LIN {X 0,Y 129.318,Z 434.565,A -85,B 0,C 180,E1 -25427.406,E2 -25427.406} C_VEL
LIN {X 0,Y 134.78,Z 442.453,A -85,B 0,C 180,E1 -25430.686,E2 -25430.686} C_VEL
LIN {X 0,Y 140.996,Z 452.81,A -85,B 0,C 180,E1 -25434.022,E2 -25434.022} C_VEL
LIN {X 0,Y 146.703,Z 463.984,A -85,B 0,C 180,E1 -25436.807,E2 -25436.807} C_VEL
LIN {X 0,Y 149.634,Z 472.659,A -85,B 0,C 180,E1 -25438.294,E2 -25438.294} C_VEL
LIN {X 0,Y 146.442,Z 521.623,A -85,B 0,C 180,E1 -25440.39,E2 -25440.39} C_VEL
LIN {X 0,Y 144.723,Z 534.957,A -85,B 0,C 180,E1 -25441.401,E2 -25441.401} C_VEL
LIN {X 0,Y 142.363,Z 547.629,A -85,B 0,C 180,E1 -25442.871,E2 -25442.871} C_VEL
LIN {X 0,Y 139.472,Z 559.922,A -85,B 0,C 180,E1 -25444.918,E2 -25444.918} C_VEL
LIN {X 0,Y 136.356,Z 570.543,A -85,B 0,C 180,E1 -25447.259,E2 -25447.259} C_VEL
LIN {X 0,Y 133.114,Z 580.026,A -85,B 0,C 180,E1 -25449.929,E2 -25449.929} C_VEL
LIN {X 0,Y 129.657,Z 589.7,A -85,B 0,C 180,E1 -25453.466,E2 -25453.466} C_VEL
LIN {X 0,Y 126.749,Z 597.618,A -85,B 0,C 180,E1 -25457.185,E2 -25457.185} C_VEL
LIN {X 0,Y 123.714,Z 605.371,A -85,B 0,C 180,E1 -25461.835,E2 -25461.835} C_VEL
LIN {X 0,Y 121.559,Z 611.578,A -85,B 0,C 180,E1 -25466.685,E2 -25466.685} C_VEL
LIN {X 0,Y 120.174,Z 616.507,A -85,B 0,C 180,E1 -25471.675,E2 -25471.675} C_VEL
LIN {X 0,Y 119.203,Z 620.325,A -85,B 0,C 180,E1 -25476.771,E2 -25476.771} C_VEL
LIN {X 0,Y 118.82,Z 622.302,A -85,B 0,C 180,E1 -25480.22,E2 -25480.22} C_VEL
LIN {X 0,Y 118.766,Z 623.841,A -85,B 0,C 180,E1 -25483.691,E2 -25483.691} C_VEL
LIN {X 0,Y 119.319,Z 625.43,A -85,B 0,C 180,E1 -25489.54,E2 -25489.54} C_VEL
LIN {X 0,Y 120.253,Z 625.873,A -85,B 0,C 180,E1 -25494.147,E2 -25494.147} C_VEL
LIN {X 0,Y 121.437,Z 625.705,A -85,B 0,C 180,E1 -25497.579,E2 -25497.579} C_VEL
LIN {X 0,Y 123.02,Z 625.088,A -85,B 0,C 180,E1 -25501.026,E2 -25501.026} C_VEL
LIN {X 0,Y 124.883,Z 624.1,A -85,B 0,C 180,E1 -25504.246,E2 -25504.246} C_VEL
LIN {X 0,Y 127.173,Z 622.663,A -85,B 0,C 180,E1 -25507.435,E2 -25507.435} C_VEL
LIN {X 0,Y 131.368,Z 619.573,A -85,B 0,C 180,E1 -25512.044,E2 -25512.044} C_VEL
LIN {X 0,Y 136.162,Z 615.452,A -85,B 0,C 180,E1 -25516.268,E2 -25516.268} C_VEL
LIN {X 0,Y 141.896,Z 609.877,A -85,B 0,C 180,E1 -25520.311,E2 -25520.311} C_VEL
LIN {X 0,Y 147.954,Z 603.18,A -85,B 0,C 180,E1 -25523.852,E2 -25523.852} C_VEL
LIN {X 0,Y 153.971,Z 595.672,A -85,B 0,C 180,E1 -25526.788,E2 -25526.788} C_VEL
LIN {X 0,Y 159.544,Z 587.649,A -85,B 0,C 180,E1 -25529.199,E2 -25529.199} C_VEL
LIN {X 0,Y 165.169,Z 578.312,A -85,B 0,C 180,E1 -25531.351,E2 -25531.351} C_VEL
LIN {X 0,Y 170.467,Z 567.735,A -85,B 0,C 180,E1 -25533.211,E2 -25533.211} C_VEL
LIN {X 0,Y 174.935,Z 556.816,A -85,B 0,C 180,E1 -25534.676,E2 -25534.676} C_VEL
LIN {X 0,Y 179.164,Z 543.992,A -85,B 0,C 180,E1 -25535.89,E2 -25535.89} C_VEL
LIN {X 0,Y 182.11,Z 531.516,A -85,B 0,C 180,E1 -25536.711,E2 -25536.711} C_VEL
LIN {X 0,Y 184.136,Z 518.177,A -85,B 0,C 180,E1 -25537.258,E2 -25537.258} C_VEL
LIN {X 0,Y 185.4,Z 503.746,A -85,B 0,C 180,E1 -25537.724,E2 -25537.724} C_VEL
LIN {X 0,Y 181.912,Z 495.534,A -85,B 0,C 180,E1 -25540.462,E2 -25540.462} C_VEL
LIN {X 0,Y 178.893,Z 489.105,A -85,B 0,C 180,E1 -25543.103,E2 -25543.103} C_VEL
LIN {X 0,Y 175.604,Z 483.621,A -85,B 0,C 180,E1 -25546.287,E2 -25546.287} C_VEL
LIN {X 0,Y 173.351,Z 479.892,A -85,B 0,C 180,E1 -25548.853,E2 -25548.853} C_VEL
LIN {X 0,Y 171.062,Z 476.076,A -85,B 0,C 180,E1 -25552.03,E2 -25552.03} C_VEL
LIN {X 0,Y 168.902,Z 472.452,A -85,B 0,C 180,E1 -25555.974,E2 -25555.974} C_VEL
LIN {X 0,Y 168.299,Z 471.765,A -85,B 0,C 180,E1 -25557.306,E2 -25557.306} C_VEL
LIN {X 0,Y 166.803,Z 469.612,A -85,B 0,C 180,E1 -25562.415,E2 -25562.415} C_VEL
LIN {X 0,Y 166.469,Z 469.381,A -85,B 0,C 180,E1 -25568.011,E2 -25568.011} C_VEL
LIN {X 0,Y 168.639,Z 472.395,A -85,B 0,C 180,E1 -25576.378,E2 -25576.378} C_VEL
LIN {X 0,Y 170.598,Z 475.906,A -85,B 0,C 180,E1 -25580.183,E2 -25580.183} C_VEL
LIN {X 0,Y 171.488,Z 476.948,A -85,B 0,C 180,E1 -25581.499,E2 -25581.499} C_VEL
LIN {X 0,Y 174.003,Z 481.404,A -85,B 0,C 180,E1 -25584.839,E2 -25584.839} C_VEL
LIN {X 0,Y 176.64,Z 486.542,A -85,B 0,C 180,E1 -25587.76,E2 -25587.76} C_VEL
LIN {X 0,Y 179.778,Z 493.205,A -85,B 0,C 180,E1 -25590.771,E2 -25590.771} C_VEL
LIN {X 0,Y 183.644,Z 502.498,A -85,B 0,C 180,E1 -25594.035,E2 -25594.035} C_VEL
LIN {X 0,Y 185.144,Z 506.515,A -85,B 0,C 180,E1 -25595.205,E2 -25595.205} C_VEL
LIN {X 0,Y 183.231,Z 526.342,A -85,B 0,C 180,E1 -25595.88,E2 -25595.88} C_VEL
LIN {X 0,Y 180.741,Z 539.674,A -85,B 0,C 180,E1 -25596.566,E2 -25596.566} C_VEL
LIN {X 0,Y 177.685,Z 550.971,A -85,B 0,C 180,E1 -25597.424,E2 -25597.424} C_VEL
LIN {X 0,Y 173.234,Z 563.127,A -85,B 0,C 180,E1 -25598.654,E2 -25598.654} C_VEL
LIN {X 0,Y 168.106,Z 574.487,A -85,B 0,C 180,E1 -25600.275,E2 -25600.275} C_VEL
LIN {X 0,Y 162.509,Z 584.748,A -85,B 0,C 180,E1 -25602.219,E2 -25602.219} C_VEL
LIN {X 0,Y 157.267,Z 593.136,A -85,B 0,C 180,E1 -25604.358,E2 -25604.358} C_VEL
LIN {X 0,Y 150.468,Z 602.273,A -85,B 0,C 180,E1 -25607.372,E2 -25607.372} C_VEL
LIN {X 0,Y 144.164,Z 609.633,A -85,B 0,C 180,E1 -25610.675,E2 -25610.675} C_VEL
LIN {X 0,Y 138.227,Z 615.973,A -85,B 0,C 180,E1 -25614.644,E2 -25614.644} C_VEL
LIN {X 0,Y 133.531,Z 620.248,A -85,B 0,C 180,E1 -25618.245,E2 -25618.245} C_VEL
LIN {X 0,Y 129.165,Z 623.859,A -85,B 0,C 180,E1 -25622.453,E2 -25622.453} C_VEL
LIN {X 0,Y 125.462,Z 626.488,A -85,B 0,C 180,E1 -25626.915,E2 -25626.915} C_VEL
LIN {X 0,Y 121.969,Z 628.597,A -85,B 0,C 180,E1 -25633.257,E2 -25633.257} C_VEL
LIN {X 0,Y 119.96,Z 629.091,A -85,B 0,C 180,E1 -25639.878,E2 -25639.878} C_VEL
LIN {X 0,Y 119.462,Z 628.772,A -85,B 0,C 180,E1 -25643.244,E2 -25643.244} C_VEL
LIN {X 0,Y 119.228,Z 628.073,A -85,B 0,C 180,E1 -25646.622,E2 -25646.622} C_VEL
LIN {X 0,Y 119.292,Z 626.945,A -85,B 0,C 180,E1 -25650.001,E2 -25650.001} C_VEL
LIN {X 0,Y 119.221,Z 625.38,A -85,B 0,C 180,E1 -25653.38,E2 -25653.38} C_VEL
LIN {X 0,Y 119.525,Z 622.215,A -85,B 0,C 180,E1 -25658.454,E2 -25658.454} C_VEL
LIN {X 0,Y 120.525,Z 617.966,A -85,B 0,C 180,E1 -25663.489,E2 -25663.489} C_VEL
LIN {X 0,Y 122.565,Z 611.486,A -85,B 0,C 180,E1 -25669.252,E2 -25669.252} C_VEL
LIN {X 0,Y 125.294,Z 604.381,A -85,B 0,C 180,E1 -25673.996,E2 -25673.996} C_VEL
LIN {X 0,Y 128.645,Z 595.462,A -85,B 0,C 180,E1 -25678.556,E2 -25678.556} C_VEL
LIN {X 0,Y 129.744,Z 592.221,A -85,B 0,C 180,E1 -25679.96,E2 -25679.96} C_VEL
LIN {X 0,Y 130.741,Z 588.009,A -85,B 0,C 180,E1 -25681.699,E2 -25681.699} C_VEL
LIN {X 0,Y 130.735,Z 580.813,A -85,B 0,C 180,E1 -25684.674,E2 -25684.674} C_VEL
LIN {X 0,Y 130.793,Z 573.141,A -85,B 0,C 180,E1 -25687.438,E2 -25687.438} C_VEL
LIN {X 0,Y 131.839,Z 568.125,A -85,B 0,C 180,E1 -25688.78,E2 -25688.78} C_VEL
LIN {X 0,Y 134.682,Z 558.276,A -85,B 0,C 180,E1 -25690.713,E2 -25690.713} C_VEL
LIN {X 0,Y 137.347,Z 546.808,A -85,B 0,C 180,E1 -25692.439,E2 -25692.439} C_VEL
LIN {X 0,Y 139.629,Z 533.737,A -85,B 0,C 180,E1 -25693.795,E2 -25693.795} C_VEL
LIN {X 0,Y 141.126,Z 520.65,A -85,B 0,C 180,E1 -25694.629,E2 -25694.629} C_VEL
LIN {X 0,Y 143.948,Z 477.532,A -85,B 0,C 180,E1 -25696.505,E2 -25696.505} C_VEL
LIN {X 0,Y 139.603,Z 464.581,A -85,B 0,C 180,E1 -25698.949,E2 -25698.949} C_VEL
LIN {X 0,Y 136.315,Z 456.813,A -85,B 0,C 180,E1 -25700.824,E2 -25700.824} C_VEL
LIN {X 0,Y 131.62,Z 448.624,A -85,B 0,C 180,E1 -25703.541,E2 -25703.541} C_VEL
LIN {X 0,Y 127.404,Z 442.333,A -85,B 0,C 180,E1 -25706.19,E2 -25706.19} C_VEL
LIN {X 0,Y 124.865,Z 438.651,A -85,B 0,C 180,E1 -25707.944,E2 -25707.944} C_VEL
LIN {X 0,Y 121.967,Z 434.646,A -85,B 0,C 180,E1 -25710.108,E2 -25710.108} C_VEL
LIN {X 0,Y 119.651,Z 431.734,A -85,B 0,C 180,E1 -25711.972,E2 -25711.972} C_VEL
LIN {X 0,Y 118.813,Z 430.199,A -85,B 0,C 180,E1 -25712.74,E2 -25712.74} C_VEL
LIN {X 0,Y 116.336,Z 428.193,A -85,B 0,C 180,E1 -25714.876,E2 -25714.876} C_VEL
LIN {X 0,Y 115.061,Z 425.271,A -85,B 0,C 180,E1 -25716.596,E2 -25716.596} C_VEL
LIN {X 0,Y 114.987,Z 424.725,A -85,B 0,C 180,E1 -25717.686,E2 -25717.686} C_VEL
LIN {X 0,Y 114.999,Z 424.63,A -85,B 0,C 180,E1 -25722.207,E2 -25722.207} C_VEL
LIN {X 0,Y 115.248,Z 424.589,A -85,B 0,C 180,E1 -25727.343,E2 -25727.343} C_VEL
LIN {X 0,Y 115.361,Z 424.586,A -85,B 0,C 180,E1 -25733.001,E2 -25733.001} C_VEL
LIN {X 0,Y 115.992,Z 424.48,A -85,B 0,C 180,E1 -25740,E2 -25740} C_VEL
LIN {X 0,Y 115.365,Z 424.614,A -85,B 0,C 180,E1 -25746.998,E2 -25746.998} C_VEL
LIN {X 0,Y 115.208,Z 424.575,A -85,B 0,C 180,E1 -25752.567,E2 -25752.567} C_VEL
LIN {X 0,Y 115.005,Z 424.657,A -85,B 0,C 180,E1 -25757.791,E2 -25757.791} C_VEL
LIN {X 0,Y 114.946,Z 424.613,A -85,B 0,C 180,E1 -25763.491,E2 -25763.491} C_VEL
LIN {X 0,Y 114.862,Z 424.646,A -85,B 0,C 180,E1 -25771.062,E2 -25771.062} C_VEL
LIN {X 0,Y 114.893,Z 424.978,A -85,B 0,C 180,E1 -25776.14,E2 -25776.14} C_VEL
LIN {X 0,Y 115.165,Z 426.179,A -85,B 0,C 180,E1 -25777.121,E2 -25777.121} C_VEL
LIN {X 0,Y 116.635,Z 428.622,A -85,B 0,C 180,E1 -25778.672,E2 -25778.672} C_VEL
LIN {X 0,Y 118.86,Z 430.392,A -85,B 0,C 180,E1 -25780.572,E2 -25780.572} C_VEL
LIN {X 0,Y 120.727,Z 433.562,A -85,B 0,C 180,E1 -25782.221,E2 -25782.221} C_VEL
LIN {X 0,Y 122.798,Z 435.75,A -85,B 0,C 180,E1 -25783.788,E2 -25783.788} C_VEL
LIN {X 0,Y 125.433,Z 439.341,A -85,B 0,C 180,E1 -25785.707,E2 -25785.707} C_VEL
LIN {X 0,Y 131.141,Z 447.832,A -85,B 0,C 180,E1 -25789.424,E2 -25789.424} C_VEL
LIN {X 0,Y 136.678,Z 457.327,A -85,B 0,C 180,E1 -25792.621,E2 -25792.621} C_VEL
LIN {X 0,Y 141.992,Z 468.051,A -85,B 0,C 180,E1 -25795.435,E2 -25795.435} C_VEL
LIN {X 0,Y 144.087,Z 474.399,A -85,B 0,C 180,E1 -25796.594,E2 -25796.594} C_VEL
LIN {X 0,Y 140.883,Z 521.133,A -85,B 0,C 180,E1 -25798.623,E2 -25798.623} C_VEL
LIN {X 0,Y 139.202,Z 534.074,A -85,B 0,C 180,E1 -25799.594,E2 -25799.594} C_VEL
LIN {X 0,Y 136.886,Z 546.091,A -85,B 0,C 180,E1 -25800.956,E2 -25800.956} C_VEL
LIN {X 0,Y 134.056,Z 558.251,A -85,B 0,C 180,E1 -25802.952,E2 -25802.952} C_VEL
LIN {X 0,Y 130.727,Z 569.365,A -85,B 0,C 180,E1 -25805.377,E2 -25805.377} C_VEL
LIN {X 0,Y 127.21,Z 579.081,A -85,B 0,C 180,E1 -25808.104,E2 -25808.104} C_VEL
LIN {X 0,Y 124.312,Z 587.125,A -85,B 0,C 180,E1 -25811.029,E2 -25811.029} C_VEL
LIN {X 0,Y 120.984,Z 595.498,A -85,B 0,C 180,E1 -25814.846,E2 -25814.846} C_VEL
LIN {X 0,Y 117.604,Z 603.695,A -85,B 0,C 180,E1 -25819.672,E2 -25819.672} C_VEL
LIN {X 0,Y 115.127,Z 610.28,A -85,B 0,C 180,E1 -25824.745,E2 -25824.745} C_VEL
LIN {X 0,Y 113.439,Z 615.521,A -85,B 0,C 180,E1 -25829.999,E2 -25829.999} C_VEL
LIN {X 0,Y 112.311,Z 619.605,A -85,B 0,C 180,E1 -25835.385,E2 -25835.385} C_VEL
LIN {X 0,Y 111.687,Z 622.638,A -85,B 0,C 180,E1 -25840.88,E2 -25840.88} C_VEL
LIN {X 0,Y 111.71,Z 624.093,A -85,B 0,C 180,E1 -25844.574,E2 -25844.574} C_VEL
LIN {X 0,Y 112.294,Z 625.509,A -85,B 0,C 180,E1 -25850.151,E2 -25850.151} C_VEL
LIN {X 0,Y 113.547,Z 625.982,A -85,B 0,C 180,E1 -25855.673,E2 -25855.673} C_VEL
LIN {X 0,Y 116.348,Z 625.237,A -85,B 0,C 180,E1 -25862.256,E2 -25862.256} C_VEL
LIN {X 0,Y 118.825,Z 624.054,A -85,B 0,C 180,E1 -25866.259,E2 -25866.259} C_VEL
LIN {X 0,Y 121.359,Z 622.53,A -85,B 0,C 180,E1 -25869.568,E2 -25869.568} C_VEL
LIN {X 0,Y 125.883,Z 619.394,A -85,B 0,C 180,E1 -25874.254,E2 -25874.254} C_VEL
LIN {X 0,Y 131.134,Z 615.125,A -85,B 0,C 180,E1 -25878.615,E2 -25878.615} C_VEL
LIN {X 0,Y 138.062,Z 608.661,A -85,B 0,C 180,E1 -25883.173,E2 -25883.173} C_VEL
LIN {X 0,Y 144.889,Z 601.318,A -85,B 0,C 180,E1 -25886.794,E2 -25886.794} C_VEL
LIN {X 0,Y 152.181,Z 592.143,A -85,B 0,C 180,E1 -25890.03,E2 -25890.03} C_VEL
LIN {X 0,Y 158.484,Z 582.794,A -85,B 0,C 180,E1 -25892.483,E2 -25892.483} C_VEL
LIN {X 0,Y 164.657,Z 571.813,A -85,B 0,C 180,E1 -25894.603,E2 -25894.603} C_VEL
LIN {X 0,Y 169.863,Z 560.436,A -85,B 0,C 180,E1 -25896.26,E2 -25896.26} C_VEL
LIN {X 0,Y 174.065,Z 549.107,A -85,B 0,C 180,E1 -25897.453,E2 -25897.453} C_VEL
LIN {X 0,Y 177.553,Z 536.548,A -85,B 0,C 180,E1 -25898.397,E2 -25898.397} C_VEL
LIN {X 0,Y 180.124,Z 522.889,A -85,B 0,C 180,E1 -25899.071,E2 -25899.071} C_VEL
LIN {X 0,Y 181.693,Z 506.768,A -85,B 0,C 180,E1 -25899.627,E2 -25899.627} C_VEL
LIN {X 0,Y 178.396,Z 498.733,A -85,B 0,C 180,E1 -25902.521,E2 -25902.521} C_VEL
LIN {X 0,Y 176.056,Z 493.796,A -85,B 0,C 180,E1 -25904.782,E2 -25904.782} C_VEL
LIN {X 0,Y 173.48,Z 489.445,A -85,B 0,C 180,E1 -25907.508,E2 -25907.508} C_VEL
LIN {X 0,Y 171.557,Z 486.149,A -85,B 0,C 180,E1 -25909.885,E2 -25909.885} C_VEL
LIN {X 0,Y 169.591,Z 482.674,A -85,B 0,C 180,E1 -25912.859,E2 -25912.859} C_VEL
LIN {X 0,Y 167.615,Z 478.978,A -85,B 0,C 180,E1 -25916.845,E2 -25916.845} C_VEL
LIN {X 0,Y 165.921,Z 476.673,A -85,B 0,C 180,E1 -25922.428,E2 -25922.428} C_VEL
LIN {X 0,Y 165.561,Z 476.29,A -85,B 0,C 180,E1 -25927.317,E2 -25927.317} C_VEL
LIN {X 0,Y 167.481,Z 479.209,A -85,B 0,C 180,E1 -25935.797,E2 -25935.797} C_VEL
LIN {X 0,Y 169.372,Z 482.752,A -85,B 0,C 180,E1 -25939.703,E2 -25939.703} C_VEL
LIN {X 0,Y 170.183,Z 483.814,A -85,B 0,C 180,E1 -25940.976,E2 -25940.976} C_VEL
LIN {X 0,Y 172.364,Z 487.944,A -85,B 0,C 180,E1 -25944.063,E2 -25944.063} C_VEL
LIN {X 0,Y 174.88,Z 493.165,A -85,B 0,C 180,E1 -25947.032,E2 -25947.032} C_VEL
LIN {X 0,Y 177.635,Z 499.469,A -85,B 0,C 180,E1 -25949.858,E2 -25949.858} C_VEL
LIN {X 0,Y 180.859,Z 507.72,A -85,B 0,C 180,E1 -25952.793,E2 -25952.793} C_VEL
LIN {X 0,Y 181.504,Z 509.556,A -85,B 0,C 180,E1 -25953.349,E2 -25953.349} C_VEL
LIN {X 0,Y 179.683,Z 527.031,A -85,B 0,C 180,E1 -25953.95,E2 -25953.95} C_VEL
LIN {X 0,Y 177.015,Z 540.483,A -85,B 0,C 180,E1 -25954.637,E2 -25954.637} C_VEL
LIN {X 0,Y 173.548,Z 552.493,A -85,B 0,C 180,E1 -25955.577,E2 -25955.577} C_VEL
LIN {X 0,Y 168.924,Z 564.343,A -85,B 0,C 180,E1 -25956.788,E2 -25956.788} C_VEL
LIN {X 0,Y 163.64,Z 575.455,A -85,B 0,C 180,E1 -25958.393,E2 -25958.393} C_VEL
LIN {X 0,Y 158.507,Z 584.464,A -85,B 0,C 180,E1 -25960.11,E2 -25960.11} C_VEL
LIN {X 0,Y 152.417,Z 593.732,A -85,B 0,C 180,E1 -25962.461,E2 -25962.461} C_VEL
LIN {X 0,Y 145.351,Z 602.724,A -85,B 0,C 180,E1 -25965.487,E2 -25965.487} C_VEL
LIN {X 0,Y 138.767,Z 609.987,A -85,B 0,C 180,E1 -25968.824,E2 -25968.824} C_VEL
LIN {X 0,Y 133.119,Z 615.582,A -85,B 0,C 180,E1 -25972.366,E2 -25972.366} C_VEL
LIN {X 0,Y 127.555,Z 620.438,A -85,B 0,C 180,E1 -25976.568,E2 -25976.568} C_VEL
LIN {X 0,Y 122.913,Z 623.977,A -85,B 0,C 180,E1 -25980.922,E2 -25980.922} C_VEL
LIN {X 0,Y 118.958,Z 626.536,A -85,B 0,C 180,E1 -25985.573,E2 -25985.573} C_VEL
LIN {X 0,Y 116.841,Z 627.752,A -85,B 0,C 180,E1 -25988.846,E2 -25988.846} C_VEL
LIN {X 0,Y 113.889,Z 628.95,A -85,B 0,C 180,E1 -25995.711,E2 -25995.711} C_VEL
LIN {X 0,Y 112.407,Z 628.623,A -85,B 0,C 180,E1 -26002.818,E2 -26002.818} C_VEL
LIN {X 0,Y 112.139,Z 627.878,A -85,B 0,C 180,E1 -26006.408,E2 -26006.408} C_VEL
LIN {X 0,Y 112.205,Z 626.699,A -85,B 0,C 180,E1 -26010.001,E2 -26010.001} C_VEL
LIN {X 0,Y 112.18,Z 624.147,A -85,B 0,C 180,E1 -26015.393,E2 -26015.393} C_VEL
LIN {X 0,Y 112.788,Z 620.563,A -85,B 0,C 180,E1 -26020.775,E2 -26020.775} C_VEL
LIN {X 0,Y 114.122,Z 615.843,A -85,B 0,C 180,E1 -26026.089,E2 -26026.089} C_VEL
LIN {X 0,Y 116.283,Z 609.846,A -85,B 0,C 180,E1 -26031.262,E2 -26031.262} C_VEL
LIN {X 0,Y 119.282,Z 602.352,A -85,B 0,C 180,E1 -26036.225,E2 -26036.225} C_VEL
LIN {X 0,Y 122.1,Z 595.407,A -85,B 0,C 180,E1 -26039.83,E2 -26039.83} C_VEL
LIN {X 0,Y 125.192,Z 587.373,A -85,B 0,C 180,E1 -26043.184,E2 -26043.184} C_VEL
LIN {X 0,Y 128.741,Z 577.497,A -85,B 0,C 180,E1 -26046.418,E2 -26046.418} C_VEL
LIN {X 0,Y 131.376,Z 569.557,A -85,B 0,C 180,E1 -26048.454,E2 -26048.454} C_VEL
LIN {X 0,Y 131.839,Z 568.125,A -85,B 0,C 180,E1 -26048.78,E2 -26048.78} C_VEL
LIN {X 0,Y 132.859,Z 563.05,A -85,B 0,C 180,E1 -26050.022,E2 -26050.022} C_VEL
LIN {X 0,Y 132.817,Z 554.574,A -85,B 0,C 180,E1 -26052.259,E2 -26052.259} C_VEL
LIN {X 0,Y 132.492,Z 545.766,A -85,B 0,C 180,E1 -26054.245,E2 -26054.245} C_VEL
LIN {X 0,Y 133.005,Z 540.169,A -85,B 0,C 180,E1 -26055.051,E2 -26055.051} C_VEL
LIN {X 0,Y 134.98,Z 527.372,A -85,B 0,C 180,E1 -26056.12,E2 -26056.12} C_VEL
LIN {X 0,Y 136.613,Z 507.055,A -85,B 0,C 180,E1 -26057.117,E2 -26057.117} C_VEL
LIN {X 0,Y 138.496,Z 479.327,A -85,B 0,C 180,E1 -26058.342,E2 -26058.342} C_VEL
LIN {X 0,Y 134.531,Z 467.157,A -85,B 0,C 180,E1 -26060.808,E2 -26060.808} C_VEL
LIN {X 0,Y 131.682,Z 460.465,A -85,B 0,C 180,E1 -26062.575,E2 -26062.575} C_VEL
LIN {X 0,Y 127.061,Z 452.375,A -85,B 0,C 180,E1 -26065.502,E2 -26065.502} C_VEL
LIN {X 0,Y 121.655,Z 444.25,A -85,B 0,C 180,E1 -26069.351,E2 -26069.351} C_VEL
LIN {X 0,Y 118.978,Z 440.456,A -85,B 0,C 180,E1 -26071.511,E2 -26071.511} C_VEL
LIN {X 0,Y 116.491,Z 436.975,A -85,B 0,C 180,E1 -26073.722,E2 -26073.722} C_VEL
LIN {X 0,Y 115.62,Z 436.086,A -85,B 0,C 180,E1 -26074.514,E2 -26074.514} C_VEL
LIN {X 0,Y 113.277,Z 433.358,A -85,B 0,C 180,E1 -26076.846,E2 -26076.846} C_VEL
LIN {X 0,Y 112.165,Z 431.206,A -85,B 0,C 180,E1 -26078.159,E2 -26078.159} C_VEL
LIN {X 0,Y 109.524,Z 429.225,A -85,B 0,C 180,E1 -26081.164,E2 -26081.164} C_VEL
LIN {X 0,Y 108.076,Z 426.18,A -85,B 0,C 180,E1 -26083.713,E2 -26083.713} C_VEL
LIN {X 0,Y 108.087,Z 425.561,A -85,B 0,C 180,E1 -26085.61,E2 -26085.61} C_VEL
LIN {X 0,Y 108.25,Z 425.449,A -85,B 0,C 180,E1 -26088.768,E2 -26088.768} C_VEL
LIN {X 0,Y 108.444,Z 425.461,A -85,B 0,C 180,E1 -26096.284,E2 -26096.284} C_VEL
LIN {X 0,Y 108.918,Z 425.36,A -85,B 0,C 180,E1 -26100,E2 -26100} C_VEL
LIN {X 0,Y 108.301,Z 425.486,A -85,B 0,C 180,E1 -26107.457,E2 -26107.457} C_VEL
LIN {X 0,Y 108.141,Z 425.454,A -85,B 0,C 180,E1 -26112.881,E2 -26112.881} C_VEL
LIN {X 0,Y 107.899,Z 425.534,A -85,B 0,C 180,E1 -26119.006,E2 -26119.006} C_VEL
LIN {X 0,Y 107.858,Z 425.495,A -85,B 0,C 180,E1 -26124.184,E2 -26124.184} C_VEL
LIN {X 0,Y 107.848,Z 425.864,A -85,B 0,C 180,E1 -26128.724,E2 -26128.724} C_VEL
LIN {X 0,Y 108.115,Z 426.85,A -85,B 0,C 180,E1 -26129.981,E2 -26129.981} C_VEL
LIN {X 0,Y 109.699,Z 429.557,A -85,B 0,C 180,E1 -26132.336,E2 -26132.336} C_VEL
LIN {X 0,Y 112.33,Z 431.61,A -85,B 0,C 180,E1 -26135.309,E2 -26135.309} C_VEL
LIN {X 0,Y 114.05,Z 434.601,A -85,B 0,C 180,E1 -26137.252,E2 -26137.252} C_VEL
LIN {X 0,Y 116.237,Z 436.761,A -85,B 0,C 180,E1 -26139.312,E2 -26139.312} C_VEL
LIN {X 0,Y 118.636,Z 440.296,A -85,B 0,C 180,E1 -26141.49,E2 -26141.49} C_VEL
LIN {X 0,Y 120.154,Z 442.185,A -85,B 0,C 180,E1 -26142.728,E2 -26142.728} C_VEL
LIN {X 0,Y 123.457,Z 446.99,A -85,B 0,C 180,E1 -26145.266,E2 -26145.266} C_VEL
LIN {X 0,Y 127.417,Z 452.926,A -85,B 0,C 180,E1 -26147.988,E2 -26147.988} C_VEL
LIN {X 0,Y 132.94,Z 462.784,A -85,B 0,C 180,E1 -26151.428,E2 -26151.428} C_VEL
LIN {X 0,Y 137.347,Z 472.094,A -85,B 0,C 180,E1 -26153.96,E2 -26153.96} C_VEL
LIN {X 0,Y 138.653,Z 476.309,A -85,B 0,C 180,E1 -26154.763,E2 -26154.763} C_VEL
LIN {X 0,Y 135.405,Z 521.455,A -85,B 0,C 180,E1 -26156.767,E2 -26156.767} C_VEL
LIN {X 0,Y 133.53,Z 534.935,A -85,B 0,C 180,E1 -26157.814,E2 -26157.814} C_VEL
LIN {X 0,Y 130.933,Z 547.734,A -85,B 0,C 180,E1 -26159.353,E2 -26159.353} C_VEL
LIN {X 0,Y 128.253,Z 558.398,A -85,B 0,C 180,E1 -26161.178,E2 -26161.178} C_VEL
LIN {X 0,Y 124.76,Z 569.487,A -85,B 0,C 180,E1 -26163.665,E2 -26163.665} C_VEL
LIN {X 0,Y 121.064,Z 579.199,A -85,B 0,C 180,E1 -26166.477,E2 -26166.477} C_VEL
LIN {X 0,Y 117.602,Z 588.138,A -85,B 0,C 180,E1 -26169.902,E2 -26169.902} C_VEL
LIN {X 0,Y 114.124,Z 596.359,A -85,B 0,C 180,E1 -26173.911,E2 -26173.911} C_VEL
LIN {X 0,Y 110.596,Z 604.428,A -85,B 0,C 180,E1 -26179.009,E2 -26179.009} C_VEL
LIN {X 0,Y 108.028,Z 610.882,A -85,B 0,C 180,E1 -26184.399,E2 -26184.399} C_VEL
LIN {X 0,Y 106.283,Z 616.003,A -85,B 0,C 180,E1 -26189.999,E2 -26189.999} C_VEL
LIN {X 0,Y 105.113,Z 619.996,A -85,B 0,C 180,E1 -26195.755,E2 -26195.755} C_VEL
LIN {X 0,Y 104.565,Z 622.949,A -85,B 0,C 180,E1 -26201.631,E2 -26201.631} C_VEL
LIN {X 0,Y 104.659,Z 624.343,A -85,B 0,C 180,E1 -26205.58,E2 -26205.58} C_VEL
LIN {X 0,Y 105.303,Z 625.592,A -85,B 0,C 180,E1 -26210.873,E2 -26210.873} C_VEL
LIN {X 0,Y 106.915,Z 626.066,A -85,B 0,C 180,E1 -26217.394,E2 -26217.394} C_VEL
LIN {X 0,Y 109.77,Z 625.379,A -85,B 0,C 180,E1 -26223.662,E2 -26223.662} C_VEL
LIN {X 0,Y 112.918,Z 623.986,A -85,B 0,C 180,E1 -26228.489,E2 -26228.489} C_VEL
LIN {X 0,Y 118.288,Z 620.802,A -85,B 0,C 180,E1 -26234.523,E2 -26234.523} C_VEL
LIN {X 0,Y 124.379,Z 616.401,A -85,B 0,C 180,E1 -26239.71,E2 -26239.71} C_VEL
LIN {X 0,Y 130.555,Z 611.225,A -85,B 0,C 180,E1 -26243.847,E2 -26243.847} C_VEL
LIN {X 0,Y 137.358,Z 604.636,A -85,B 0,C 180,E1 -26247.586,E2 -26247.586} C_VEL
LIN {X 0,Y 144.873,Z 596.194,A -85,B 0,C 180,E1 -26250.98,E2 -26250.98} C_VEL
LIN {X 0,Y 151.194,Z 587.844,A -85,B 0,C 180,E1 -26253.479,E2 -26253.479} C_VEL
LIN {X 0,Y 157.279,Z 578.52,A -85,B 0,C 180,E1 -26255.564,E2 -26255.564} C_VEL
LIN {X 0,Y 163.275,Z 567.273,A -85,B 0,C 180,E1 -26257.474,E2 -26257.474} C_VEL
LIN {X 0,Y 168.466,Z 555.235,A -85,B 0,C 180,E1 -26258.972,E2 -26258.972} C_VEL
LIN {X 0,Y 172.645,Z 542.83,A -85,B 0,C 180,E1 -26260.035,E2 -26260.035} C_VEL
LIN {X 0,Y 175.824,Z 529.456,A -85,B 0,C 180,E1 -26260.826,E2 -26260.826} C_VEL
LIN {X 0,Y 177.694,Z 516.827,A -85,B 0,C 180,E1 -26261.292,E2 -26261.292} C_VEL
LIN {X 0,Y 178.241,Z 509.938,A -85,B 0,C 180,E1 -26261.567,E2 -26261.567} C_VEL
LIN {X 0,Y 174.903,Z 501.663,A -85,B 0,C 180,E1 -26264.863,E2 -26264.863} C_VEL
LIN {X 0,Y 172.071,Z 496.371,A -85,B 0,C 180,E1 -26267.985,E2 -26267.985} C_VEL
LIN {X 0,Y 169.997,Z 492.646,A -85,B 0,C 180,E1 -26270.706,E2 -26270.706} C_VEL
LIN {X 0,Y 168.16,Z 489.241,A -85,B 0,C 180,E1 -26273.702,E2 -26273.702} C_VEL
LIN {X 0,Y 166.401,Z 485.805,A -85,B 0,C 180,E1 -26277.58,E2 -26277.58} C_VEL
LIN {X 0,Y 164.931,Z 483.64,A -85,B 0,C 180,E1 -26283.054,E2 -26283.054} C_VEL
LIN {X 0,Y 164.696,Z 483.455,A -85,B 0,C 180,E1 -26287.727,E2 -26287.727} C_VEL
LIN {X 0,Y 166.428,Z 486.28,A -85,B 0,C 180,E1 -26295.46,E2 -26295.46} C_VEL
LIN {X 0,Y 168.517,Z 489.994,A -85,B 0,C 180,E1 -26299.807,E2 -26299.807} C_VEL
LIN {X 0,Y 170.509,Z 493.899,A -85,B 0,C 180,E1 -26302.922,E2 -26302.922} C_VEL
LIN {X 0,Y 172.828,Z 499.08,A -85,B 0,C 180,E1 -26305.915,E2 -26305.915} C_VEL
LIN {X 0,Y 175.236,Z 504.883,A -85,B 0,C 180,E1 -26308.599,E2 -26308.599} C_VEL
LIN {X 0,Y 178.071,Z 512.589,A -85,B 0,C 180,E1 -26311.418,E2 -26311.418} C_VEL
LIN {X 0,Y 176.265,Z 528.184,A -85,B 0,C 180,E1 -26311.954,E2 -26311.954} C_VEL
LIN {X 0,Y 173.807,Z 540.088,A -85,B 0,C 180,E1 -26312.568,E2 -26312.568} C_VEL
LIN {X 0,Y 170.575,Z 551.119,A -85,B 0,C 180,E1 -26313.364,E2 -26313.364} C_VEL
LIN {X 0,Y 166.22,Z 562.437,A -85,B 0,C 180,E1 -26314.467,E2 -26314.467} C_VEL
LIN {X 0,Y 161.387,Z 572.607,A -85,B 0,C 180,E1 -26315.802,E2 -26315.802} C_VEL
LIN {X 0,Y 155.381,Z 583.147,A -85,B 0,C 180,E1 -26317.673,E2 -26317.673} C_VEL
LIN {X 0,Y 148.963,Z 592.656,A -85,B 0,C 180,E1 -26319.947,E2 -26319.947} C_VEL
LIN {X 0,Y 142.768,Z 600.474,A -85,B 0,C 180,E1 -26322.407,E2 -26322.407} C_VEL
LIN {X 0,Y 135.748,Z 608.136,A -85,B 0,C 180,E1 -26325.661,E2 -26325.661} C_VEL
LIN {X 0,Y 129.319,Z 614.296,A -85,B 0,C 180,E1 -26329.298,E2 -26329.298} C_VEL
LIN {X 0,Y 123.553,Z 619.21,A -85,B 0,C 180,E1 -26333.328,E2 -26333.328} C_VEL
LIN {X 0,Y 118.286,Z 623.033,A -85,B 0,C 180,E1 -26337.676,E2 -26337.676} C_VEL
LIN {X 0,Y 112.531,Z 626.584,A -85,B 0,C 180,E1 -26344.078,E2 -26344.078} C_VEL
LIN {X 0,Y 110.223,Z 627.754,A -85,B 0,C 180,E1 -26347.508,E2 -26347.508} C_VEL
LIN {X 0,Y 106.998,Z 628.865,A -85,B 0,C 180,E1 -26354.769,E2 -26354.769} C_VEL
LIN {X 0,Y 105.348,Z 628.472,A -85,B 0,C 180,E1 -26362.334,E2 -26362.334} C_VEL
LIN {X 0,Y 105.074,Z 627.665,A -85,B 0,C 180,E1 -26366.166,E2 -26366.166} C_VEL
LIN {X 0,Y 105.109,Z 626.45,A -85,B 0,C 180,E1 -26370.001,E2 -26370.001} C_VEL
LIN {X 0,Y 105.1,Z 623.828,A -85,B 0,C 180,E1 -26375.758,E2 -26375.758} C_VEL
LIN {X 0,Y 105.809,Z 620.17,A -85,B 0,C 180,E1 -26381.495,E2 -26381.495} C_VEL
LIN {X 0,Y 107.276,Z 615.369,A -85,B 0,C 180,E1 -26387.147,E2 -26387.147} C_VEL
LIN {X 0,Y 109.68,Z 609.287,A -85,B 0,C 180,E1 -26392.611,E2 -26392.611} C_VEL
LIN {X 0,Y 112.923,Z 601.693,A -85,B 0,C 180,E1 -26397.826,E2 -26397.826} C_VEL
LIN {X 0,Y 115.336,Z 596.194,A -85,B 0,C 180,E1 -26400.813,E2 -26400.813} C_VEL
LIN {X 0,Y 118.467,Z 588.438,A -85,B 0,C 180,E1 -26404.304,E2 -26404.304} C_VEL
LIN {X 0,Y 122.607,Z 577.614,A -85,B 0,C 180,E1 -26408.04,E2 -26408.04} C_VEL
LIN {X 0,Y 125.378,Z 569.721,A -85,B 0,C 180,E1 -26410.138,E2 -26410.138} C_VEL
LIN {X 0,Y 128.836,Z 558.501,A -85,B 0,C 180,E1 -26412.458,E2 -26412.458} C_VEL
LIN {X 0,Y 131.866,Z 545.924,A -85,B 0,C 180,E1 -26414.388,E2 -26414.388} C_VEL
LIN {X 0,Y 133.005,Z 540.169,A -85,B 0,C 180,E1 -26415.051,E2 -26415.051} C_VEL
LIN {X 0,Y 133.503,Z 534.504,A -85,B 0,C 180,E1 -26415.76,E2 -26415.76} C_VEL
LIN {X 0,Y 132.61,Z 525.233,A -85,B 0,C 180,E1 -26417.228,E2 -26417.228} C_VEL
LIN {X 0,Y 131.26,Z 515.868,A -85,B 0,C 180,E1 -26418.55,E2 -26418.55} C_VEL
LIN {X 0,Y 131.152,Z 510.046,A -85,B 0,C 180,E1 -26419.018,E2 -26419.018} C_VEL
LIN {X 0,Y 133.249,Z 481.15,A -85,B 0,C 180,E1 -26420.303,E2 -26420.303} C_VEL
LIN {X 0,Y 129.621,Z 469.922,A -85,B 0,C 180,E1 -26422.779,E2 -26422.779} C_VEL
LIN {X 0,Y 127.321,Z 464.542,A -85,B 0,C 180,E1 -26424.335,E2 -26424.335} C_VEL
LIN {X 0,Y 123.574,Z 457.729,A -85,B 0,C 180,E1 -26426.932,E2 -26426.932} C_VEL
LIN {X 0,Y 118.417,Z 449.676,A -85,B 0,C 180,E1 -26430.929,E2 -26430.929} C_VEL
LIN {X 0,Y 116.119,Z 446.324,A -85,B 0,C 180,E1 -26432.942,E2 -26432.942} C_VEL
LIN {X 0,Y 113.339,Z 442.451,A -85,B 0,C 180,E1 -26435.631,E2 -26435.631} C_VEL
LIN {X 0,Y 110.806,Z 439.317,A -85,B 0,C 180,E1 -26438.366,E2 -26438.366} C_VEL
LIN {X 0,Y 109.796,Z 437.594,A -85,B 0,C 180,E1 -26439.631,E2 -26439.631} C_VEL
LIN {X 0,Y 107.27,Z 435.193,A -85,B 0,C 180,E1 -26442.852,E2 -26442.852} C_VEL
LIN {X 0,Y 105.723,Z 432.295,A -85,B 0,C 180,E1 -26445.394,E2 -26445.394} C_VEL
LIN {X 0,Y 102.433,Z 429.494,A -85,B 0,C 180,E1 -26451.616,E2 -26451.616} C_VEL
LIN {X 0,Y 101.453,Z 426.975,A -85,B 0,C 180,E1 -26455.53,E2 -26455.53} C_VEL
LIN {X 0,Y 101.845,Z 426.274,A -85,B 0,C 180,E1 -26460,E2 -26460} C_VEL
LIN {X 0,Y 101.233,Z 426.38,A -85,B 0,C 180,E1 -26467.981,E2 -26467.981} C_VEL
LIN {X 0,Y 101.094,Z 426.479,A -85,B 0,C 180,E1 -26473.277,E2 -26473.277} C_VEL
LIN {X 0,Y 101.05,Z 427.365,A -85,B 0,C 180,E1 -26477.192,E2 -26477.192} C_VEL
LIN {X 0,Y 102.682,Z 430.341,A -85,B 0,C 180,E1 -26482.378,E2 -26482.378} C_VEL
LIN {X 0,Y 105.911,Z 432.777,A -85,B 0,C 180,E1 -26488.216,E2 -26488.216} C_VEL
LIN {X 0,Y 107.79,Z 436.029,A -85,B 0,C 180,E1 -26491.166,E2 -26491.166} C_VEL
LIN {X 0,Y 110.103,Z 438.116,A -85,B 0,C 180,E1 -26494.015,E2 -26494.015} C_VEL
LIN {X 0,Y 112.313,Z 441.498,A -85,B 0,C 180,E1 -26496.602,E2 -26496.602} C_VEL
LIN {X 0,Y 113.702,Z 443.031,A -85,B 0,C 180,E1 -26498.004,E2 -26498.004} C_VEL
LIN {X 0,Y 116.426,Z 446.806,A -85,B 0,C 180,E1 -26500.597,E2 -26500.597} C_VEL
LIN {X 0,Y 120.136,Z 452.36,A -85,B 0,C 180,E1 -26503.739,E2 -26503.739} C_VEL
LIN {X 0,Y 124.046,Z 458.567,A -85,B 0,C 180,E1 -26506.666,E2 -26506.666} C_VEL
LIN {X 0,Y 129.066,Z 467.882,A -85,B 0,C 180,E1 -26510.052,E2 -26510.052} C_VEL
LIN {X 0,Y 132.711,Z 475.864,A -85,B 0,C 180,E1 -26512.324,E2 -26512.324} C_VEL
LIN {X 0,Y 133.383,Z 478.193,A -85,B 0,C 180,E1 -26512.787,E2 -26512.787} C_VEL
LIN {X 0,Y 130.099,Z 521.596,A -85,B 0,C 180,E1 -26514.745,E2 -26514.745} C_VEL
LIN {X 0,Y 128.133,Z 535.026,A -85,B 0,C 180,E1 -26515.799,E2 -26515.799} C_VEL
LIN {X 0,Y 125.335,Z 548.223,A -85,B 0,C 180,E1 -26517.423,E2 -26517.423} C_VEL
LIN {X 0,Y 122.372,Z 559.187,A -85,B 0,C 180,E1 -26519.356,E2 -26519.356} C_VEL
LIN {X 0,Y 118.403,Z 570.913,A -85,B 0,C 180,E1 -26522.132,E2 -26522.132} C_VEL
LIN {X 0,Y 114.622,Z 580.385,A -85,B 0,C 180,E1 -26525.068,E2 -26525.068} C_VEL
LIN {X 0,Y 110.914,Z 589.154,A -85,B 0,C 180,E1 -26528.632,E2 -26528.632} C_VEL
LIN {X 0,Y 107.31,Z 597.219,A -85,B 0,C 180,E1 -26532.859,E2 -26532.859} C_VEL
LIN {X 0,Y 103.611,Z 605.142,A -85,B 0,C 180,E1 -26538.258,E2 -26538.258} C_VEL
LIN {X 0,Y 100.935,Z 611.448,A -85,B 0,C 180,E1 -26544.004,E2 -26544.004} C_VEL
LIN {X 0,Y 99.127,Z 616.471,A -85,B 0,C 180,E1 -26549.999,E2 -26549.999} C_VEL
LIN {X 0,Y 97.926,Z 620.375,A -85,B 0,C 180,E1 -26556.179,E2 -26556.179} C_VEL
LIN {X 0,Y 97.444,Z 623.241,A -85,B 0,C 180,E1 -26562.495,E2 -26562.495} C_VEL
LIN {X 0,Y 97.648,Z 624.594,A -85,B 0,C 180,E1 -26566.73,E2 -26566.73} C_VEL
LIN {X 0,Y 98.304,Z 625.668,A -85,B 0,C 180,E1 -26571.658,E2 -26571.658} C_VEL
LIN {X 0,Y 100.387,Z 626.149,A -85,B 0,C 180,E1 -26579.343,E2 -26579.343} C_VEL
LIN {X 0,Y 103.241,Z 625.528,A -85,B 0,C 180,E1 -26585.226,E2 -26585.226} C_VEL
LIN {X 0,Y 107.194,Z 623.901,A -85,B 0,C 180,E1 -26590.965,E2 -26590.965} C_VEL
LIN {X 0,Y 112.441,Z 621.033,A -85,B 0,C 180,E1 -26596.565,E2 -26596.565} C_VEL
LIN {X 0,Y 119.711,Z 616.137,A -85,B 0,C 180,E1 -26602.422,E2 -26602.422} C_VEL
LIN {X 0,Y 126.321,Z 610.838,A -85,B 0,C 180,E1 -26606.565,E2 -26606.565} C_VEL
LIN {X 0,Y 133.554,Z 604.108,A -85,B 0,C 180,E1 -26610.256,E2 -26610.256} C_VEL
LIN {X 0,Y 141.317,Z 595.7,A -85,B 0,C 180,E1 -26613.528,E2 -26613.528} C_VEL
LIN {X 0,Y 148.057,Z 587.03,A -85,B 0,C 180,E1 -26616.026,E2 -26616.026} C_VEL
LIN {X 0,Y 155.095,Z 576.237,A -85,B 0,C 180,E1 -26618.265,E2 -26618.265} C_VEL
LIN {X 0,Y 160.83,Z 565.458,A -85,B 0,C 180,E1 -26619.961,E2 -26619.961} C_VEL
LIN {X 0,Y 165.982,Z 553.447,A -85,B 0,C 180,E1 -26621.328,E2 -26621.328} C_VEL
LIN {X 0,Y 170.277,Z 540.291,A -85,B 0,C 180,E1 -26622.357,E2 -26622.357} C_VEL
LIN {X 0,Y 173.218,Z 527.507,A -85,B 0,C 180,E1 -26623.031,E2 -26623.031} C_VEL
LIN {X 0,Y 175.037,Z 513.44,A -85,B 0,C 180,E1 -26623.519,E2 -26623.519} C_VEL
LIN {X 0,Y 172.44,Z 506.772,A -85,B 0,C 180,E1 -26626.372,E2 -26626.372} C_VEL
LIN {X 0,Y 169.769,Z 501.64,A -85,B 0,C 180,E1 -26629.641,E2 -26629.641} C_VEL
LIN {X 0,Y 168.246,Z 498.738,A -85,B 0,C 180,E1 -26631.896,E2 -26631.896} C_VEL
LIN {X 0,Y 166.848,Z 495.904,A -85,B 0,C 180,E1 -26634.41,E2 -26634.41} C_VEL
LIN {X 0,Y 165.332,Z 492.738,A -85,B 0,C 180,E1 -26638.021,E2 -26638.021} C_VEL
LIN {X 0,Y 163.964,Z 490.591,A -85,B 0,C 180,E1 -26643.687,E2 -26643.687} C_VEL
LIN {X 0,Y 163.836,Z 490.644,A -85,B 0,C 180,E1 -26648.141,E2 -26648.141} C_VEL
LIN {X 0,Y 165.324,Z 493.156,A -85,B 0,C 180,E1 -26654.935,E2 -26654.935} C_VEL
LIN {X 0,Y 167.581,Z 497.494,A -85,B 0,C 180,E1 -26659.843,E2 -26659.843} C_VEL
LIN {X 0,Y 168.951,Z 500.415,A -85,B 0,C 180,E1 -26662.102,E2 -26662.102} C_VEL
LIN {X 0,Y 171.075,Z 505.501,A -85,B 0,C 180,E1 -26665.063,E2 -26665.063} C_VEL
LIN {X 0,Y 173.348,Z 511.506,A -85,B 0,C 180,E1 -26667.795,E2 -26667.795} C_VEL
LIN {X 0,Y 174.809,Z 515.821,A -85,B 0,C 180,E1 -26669.404,E2 -26669.404} C_VEL
LIN {X 0,Y 173.077,Z 529.377,A -85,B 0,C 180,E1 -26669.897,E2 -26669.897} C_VEL
LIN {X 0,Y 170.116,Z 542.259,A -85,B 0,C 180,E1 -26670.566,E2 -26670.566} C_VEL
LIN {X 0,Y 165.813,Z 555.47,A -85,B 0,C 180,E1 -26671.597,E2 -26671.597} C_VEL
LIN {X 0,Y 160.884,Z 566.778,A -85,B 0,C 180,E1 -26672.767,E2 -26672.767} C_VEL
LIN {X 0,Y 155.294,Z 577.303,A -85,B 0,C 180,E1 -26674.321,E2 -26674.321} C_VEL
LIN {X 0,Y 148.446,Z 587.911,A -85,B 0,C 180,E1 -26676.407,E2 -26676.407} C_VEL
LIN {X 0,Y 141.994,Z 596.523,A -85,B 0,C 180,E1 -26678.783,E2 -26678.783} C_VEL
LIN {X 0,Y 135.644,Z 603.667,A -85,B 0,C 180,E1 -26681.301,E2 -26681.301} C_VEL
LIN {X 0,Y 128.432,Z 610.711,A -85,B 0,C 180,E1 -26684.655,E2 -26684.655} C_VEL
LIN {X 0,Y 121.431,Z 616.719,A -85,B 0,C 180,E1 -26688.799,E2 -26688.799} C_VEL
LIN {X 0,Y 115.989,Z 620.797,A -85,B 0,C 180,E1 -26692.707,E2 -26692.707} C_VEL
LIN {X 0,Y 112.336,Z 623.157,A -85,B 0,C 180,E1 -26695.734,E2 -26695.734} C_VEL
LIN {X 0,Y 106.194,Z 626.634,A -85,B 0,C 180,E1 -26702.404,E2 -26702.404} C_VEL
LIN {X 0,Y 103.674,Z 627.738,A -85,B 0,C 180,E1 -26706.002,E2 -26706.002} C_VEL
LIN {X 0,Y 100.149,Z 628.781,A -85,B 0,C 180,E1 -26713.699,E2 -26713.699} C_VEL
LIN {X 0,Y 99.019,Z 628.74,A -85,B 0,C 180,E1 -26717.707,E2 -26717.707} C_VEL
LIN {X 0,Y 98.311,Z 628.305,A -85,B 0,C 180,E1 -26721.781,E2 -26721.781} C_VEL
LIN {X 0,Y 98,Z 627.449,A -85,B 0,C 180,E1 -26725.889,E2 -26725.889} C_VEL
LIN {X 0,Y 98.008,Z 626.201,A -85,B 0,C 180,E1 -26730.001,E2 -26730.001} C_VEL
LIN {X 0,Y 98.044,Z 623.509,A -85,B 0,C 180,E1 -26736.173,E2 -26736.173} C_VEL
LIN {X 0,Y 98.827,Z 619.776,A -85,B 0,C 180,E1 -26742.319,E2 -26742.319} C_VEL
LIN {X 0,Y 100.477,Z 614.896,A -85,B 0,C 180,E1 -26748.347,E2 -26748.347} C_VEL
LIN {X 0,Y 103.144,Z 608.727,A -85,B 0,C 180,E1 -26754.132,E2 -26754.132} C_VEL
LIN {X 0,Y 106.674,Z 601.028,A -85,B 0,C 180,E1 -26759.612,E2 -26759.612} C_VEL
LIN {X 0,Y 109.58,Z 594.397,A -85,B 0,C 180,E1 -26763.294,E2 -26763.294} C_VEL
LIN {X 0,Y 113.473,Z 585.554,A -85,B 0,C 180,E1 -26767.148,E2 -26767.148} C_VEL
LIN {X 0,Y 117.457,Z 575.248,A -85,B 0,C 180,E1 -26770.594,E2 -26770.594} C_VEL
LIN {X 0,Y 121.56,Z 563.843,A -85,B 0,C 180,E1 -26773.358,E2 -26773.358} C_VEL
LIN {X 0,Y 124.993,Z 551.954,A -85,B 0,C 180,E1 -26775.511,E2 -26775.511} C_VEL
LIN {X 0,Y 127.728,Z 539.321,A -85,B 0,C 180,E1 -26777.141,E2 -26777.141} C_VEL
LIN {X 0,Y 129.797,Z 526.072,A -85,B 0,C 180,E1 -26778.23,E2 -26778.23} C_VEL
LIN {X 0,Y 131.152,Z 510.046,A -85,B 0,C 180,E1 -26779.018,E2 -26779.018} C_VEL
LIN {X 0,Y 131.108,Z 500.271,A -85,B 0,C 180,E1 -26779.769,E2 -26779.769} C_VEL
LIN {X 0,Y 130.493,Z 494.552,A -85,B 0,C 180,E1 -26780.465,E2 -26780.465} C_VEL
LIN {X 0,Y 129.125,Z 487.146,A -85,B 0,C 180,E1 -26781.641,E2 -26781.641} C_VEL
LIN {X 0,Y 127.275,Z 480.06,A -85,B 0,C 180,E1 -26783.071,E2 -26783.071} C_VEL
LIN {X 0,Y 124.239,Z 470.973,A -85,B 0,C 180,E1 -26785.381,E2 -26785.381} C_VEL
LIN {X 0,Y 120.294,Z 463.248,A -85,B 0,C 180,E1 -26788.351,E2 -26788.351} C_VEL
LIN {X 0,Y 115.16,Z 454.941,A -85,B 0,C 180,E1 -26792.699,E2 -26792.699} C_VEL
LIN {X 0,Y 112.756,Z 451.374,A -85,B 0,C 180,E1 -26795.028,E2 -26795.028} C_VEL
LIN {X 0,Y 110.807,Z 448.511,A -85,B 0,C 180,E1 -26797.117,E2 -26797.117} C_VEL
LIN {X 0,Y 108.237,Z 444.911,A -85,B 0,C 180,E1 -26800.207,E2 -26800.207} C_VEL
LIN {X 0,Y 107.294,Z 443.733,A -85,B 0,C 180,E1 -26801.439,E2 -26801.439} C_VEL
LIN {X 0,Y 104.938,Z 440.855,A -85,B 0,C 180,E1 -26804.884,E2 -26804.884} C_VEL
LIN {X 0,Y 104.011,Z 438.971,A -85,B 0,C 180,E1 -26806.595,E2 -26806.595} C_VEL
LIN {X 0,Y 101.049,Z 436.17,A -85,B 0,C 180,E1 -26812.758,E2 -26812.758} C_VEL
LIN {X 0,Y 99.868,Z 433.549,A -85,B 0,C 180,E1 -26816.974,E2 -26816.974} C_VEL
LIN {X 0,Y 99.213,Z 432.88,A -85,B 0,C 180,E1 -26820,E2 -26820} C_VEL
LIN {X 0,Y 99.098,Z 433.273,A -85,B 0,C 180,E1 -26832.916,E2 -26832.916} C_VEL
LIN {X 0,Y 99.804,Z 434.23,A -85,B 0,C 180,E1 -26836.36,E2 -26836.36} C_VEL
LIN {X 0,Y 101.39,Z 437.164,A -85,B 0,C 180,E1 -26841.551,E2 -26841.551} C_VEL
LIN {X 0,Y 104.178,Z 439.481,A -85,B 0,C 180,E1 -26847.022,E2 -26847.022} C_VEL
LIN {X 0,Y 106.123,Z 442.732,A -85,B 0,C 180,E1 -26850.261,E2 -26850.261} C_VEL
LIN {X 0,Y 108.005,Z 444.653,A -85,B 0,C 180,E1 -26852.755,E2 -26852.755} C_VEL
LIN {X 0,Y 110.375,Z 448.085,A -85,B 0,C 180,E1 -26855.674,E2 -26855.674} C_VEL
LIN {X 0,Y 111.719,Z 450.051,A -85,B 0,C 180,E1 -26857.166,E2 -26857.166} C_VEL
LIN {X 0,Y 114.774,Z 454.414,A -85,B 0,C 180,E1 -26860.204,E2 -26860.204} C_VEL
LIN {X 0,Y 118.965,Z 461.058,A -85,B 0,C 180,E1 -26863.853,E2 -26863.853} C_VEL
LIN {X 0,Y 123.285,Z 468.923,A -85,B 0,C 180,E1 -26867.175,E2 -26867.175} C_VEL
LIN {X 0,Y 128.086,Z 479.316,A -85,B 0,C 180,E1 -26870.513,E2 -26870.513} C_VEL
LIN {X 0,Y 128.31,Z 480.585,A -85,B 0,C 180,E1 -26870.72,E2 -26870.72} C_VEL
LIN {X 0,Y 124.822,Z 522.625,A -85,B 0,C 180,E1 -26872.61,E2 -26872.61} C_VEL
LIN {X 0,Y 122.682,Z 536.264,A -85,B 0,C 180,E1 -26873.735,E2 -26873.735} C_VEL
LIN {X 0,Y 119.801,Z 549.044,A -85,B 0,C 180,E1 -26875.38,E2 -26875.38} C_VEL
LIN {X 0,Y 116.328,Z 560.873,A -85,B 0,C 180,E1 -26877.575,E2 -26877.575} C_VEL
LIN {X 0,Y 112.116,Z 572.318,A -85,B 0,C 180,E1 -26880.419,E2 -26880.419} C_VEL
LIN {X 0,Y 108.683,Z 580.482,A -85,B 0,C 180,E1 -26883.085,E2 -26883.085} C_VEL
LIN {X 0,Y 104.301,Z 590.154,A -85,B 0,C 180,E1 -26887.204,E2 -26887.204} C_VEL
LIN {X 0,Y 100.542,Z 598.067,A -85,B 0,C 180,E1 -26891.665,E2 -26891.665} C_VEL
LIN {X 0,Y 96.656,Z 605.808,A -85,B 0,C 180,E1 -26897.4,E2 -26897.4} C_VEL
LIN {X 0,Y 93.835,Z 612.008,A -85,B 0,C 180,E1 -26903.548,E2 -26903.548} C_VEL
LIN {X 0,Y 91.953,Z 616.935,A -85,B 0,C 180,E1 -26909.999,E2 -26909.999} C_VEL
LIN {X 0,Y 90.733,Z 620.75,A -85,B 0,C 180,E1 -26916.671,E2 -26916.671} C_VEL
LIN {X 0,Y 90.345,Z 623.531,A -85,B 0,C 180,E1 -26923.494,E2 -26923.494} C_VEL
LIN {X 0,Y 90.648,Z 624.842,A -85,B 0,C 180,E1 -26928.065,E2 -26928.065} C_VEL
LIN {X 0,Y 91.328,Z 625.746,A -85,B 0,C 180,E1 -26932.628,E2 -26932.628} C_VEL
LIN {X 0,Y 92.41,Z 626.193,A -85,B 0,C 180,E1 -26937.148,E2 -26937.148} C_VEL
LIN {X 0,Y 94.004,Z 626.232,A -85,B 0,C 180,E1 -26941.554,E2 -26941.554} C_VEL
LIN {X 0,Y 96.812,Z 625.676,A -85,B 0,C 180,E1 -26947.01,E2 -26947.01} C_VEL
LIN {X 0,Y 101.694,Z 623.818,A -85,B 0,C 180,E1 -26953.714,E2 -26953.714} C_VEL
LIN {X 0,Y 106.775,Z 621.256,A -85,B 0,C 180,E1 -26958.837,E2 -26958.837} C_VEL
LIN {X 0,Y 113.138,Z 617.341,A -85,B 0,C 180,E1 -26963.853,E2 -26963.853} C_VEL
LIN {X 0,Y 120.171,Z 612.219,A -85,B 0,C 180,E1 -26968.241,E2 -26968.241} C_VEL
LIN {X 0,Y 127.433,Z 606.043,A -85,B 0,C 180,E1 -26971.93,E2 -26971.93} C_VEL
LIN {X 0,Y 134.675,Z 598.926,A -85,B 0,C 180,E1 -26974.952,E2 -26974.952} C_VEL
LIN {X 0,Y 142.371,Z 589.903,A -85,B 0,C 180,E1 -26977.75,E2 -26977.75} C_VEL
LIN {X 0,Y 149.583,Z 579.85,A -85,B 0,C 180,E1 -26979.992,E2 -26979.992} C_VEL
LIN {X 0,Y 155.49,Z 569.927,A -85,B 0,C 180,E1 -26981.65,E2 -26981.65} C_VEL
LIN {X 0,Y 160.736,Z 559.129,A -85,B 0,C 180,E1 -26983.024,E2 -26983.024} C_VEL
LIN {X 0,Y 165.334,Z 547.261,A -85,B 0,C 180,E1 -26984.074,E2 -26984.074} C_VEL
LIN {X 0,Y 168.943,Z 534.677,A -85,B 0,C 180,E1 -26984.88,E2 -26984.88} C_VEL
LIN {X 0,Y 171.328,Z 522.385,A -85,B 0,C 180,E1 -26985.4,E2 -26985.4} C_VEL
LIN {X 0,Y 172.011,Z 517.01,A -85,B 0,C 180,E1 -26985.557,E2 -26985.557} C_VEL
LIN {X 0,Y 170.204,Z 512.191,A -85,B 0,C 180,E1 -26987.783,E2 -26987.783} C_VEL
LIN {X 0,Y 167.771,Z 507.22,A -85,B 0,C 180,E1 -26991.114,E2 -26991.114} C_VEL
LIN {X 0,Y 165.565,Z 502.562,A -85,B 0,C 180,E1 -26995.13,E2 -26995.13} C_VEL
LIN {X 0,Y 164.273,Z 499.664,A -85,B 0,C 180,E1 -26998.468,E2 -26998.468} C_VEL
LIN {X 0,Y 163.083,Z 497.642,A -85,B 0,C 180,E1 -27003.707,E2 -27003.707} C_VEL
LIN {X 0,Y 162.938,Z 497.612,A -85,B 0,C 180,E1 -27007.753,E2 -27007.753} C_VEL
LIN {X 0,Y 164.236,Z 500.021,A -85,B 0,C 180,E1 -27014.403,E2 -27014.403} C_VEL
LIN {X 0,Y 166.236,Z 504.168,A -85,B 0,C 180,E1 -27019.126,E2 -27019.126} C_VEL
LIN {X 0,Y 167.371,Z 506.81,A -85,B 0,C 180,E1 -27021.172,E2 -27021.172} C_VEL
LIN {X 0,Y 169.441,Z 512.139,A -85,B 0,C 180,E1 -27024.304,E2 -27024.304} C_VEL
LIN {X 0,Y 171.599,Z 518.628,A -85,B 0,C 180,E1 -27027.124,E2 -27027.124} C_VEL
LIN {X 0,Y 171.77,Z 519.429,A -85,B 0,C 180,E1 -27027.378,E2 -27027.378} C_VEL
LIN {X 0,Y 169.571,Z 532.971,A -85,B 0,C 180,E1 -27027.871,E2 -27027.871} C_VEL
LIN {X 0,Y 166.498,Z 544.906,A -85,B 0,C 180,E1 -27028.526,E2 -27028.526} C_VEL
LIN {X 0,Y 162.276,Z 556.88,A -85,B 0,C 180,E1 -27029.476,E2 -27029.476} C_VEL
LIN {X 0,Y 156.439,Z 569.302,A -85,B 0,C 180,E1 -27030.778,E2 -27030.778} C_VEL
LIN {X 0,Y 150.012,Z 580.508,A -85,B 0,C 180,E1 -27032.513,E2 -27032.513} C_VEL
LIN {X 0,Y 143.035,Z 590.433,A -85,B 0,C 180,E1 -27034.616,E2 -27034.616} C_VEL
LIN {X 0,Y 134.997,Z 600.055,A -85,B 0,C 180,E1 -27037.449,E2 -27037.449} C_VEL
LIN {X 0,Y 127.24,Z 607.776,A -85,B 0,C 180,E1 -27040.585,E2 -27040.585} C_VEL
LIN {X 0,Y 121.17,Z 613.045,A -85,B 0,C 180,E1 -27043.532,E2 -27043.532} C_VEL
LIN {X 0,Y 114.549,Z 618.185,A -85,B 0,C 180,E1 -27047.556,E2 -27047.556} C_VEL
LIN {X 0,Y 108.436,Z 622.198,A -85,B 0,C 180,E1 -27051.998,E2 -27051.998} C_VEL
LIN {X 0,Y 103.094,Z 625.186,A -85,B 0,C 180,E1 -27056.952,E2 -27056.952} C_VEL
LIN {X 0,Y 99.936,Z 626.671,A -85,B 0,C 180,E1 -27060.512,E2 -27060.512} C_VEL
LIN {X 0,Y 97.208,Z 627.723,A -85,B 0,C 180,E1 -27064.293,E2 -27064.293} C_VEL
LIN {X 0,Y 93.348,Z 628.697,A -85,B 0,C 180,E1 -27072.475,E2 -27072.475} C_VEL
LIN {X 0,Y 92.086,Z 628.619,A -85,B 0,C 180,E1 -27076.766,E2 -27076.766} C_VEL
LIN {X 0,Y 91.297,Z 628.122,A -85,B 0,C 180,E1 -27081.145,E2 -27081.145} C_VEL
LIN {X 0,Y 90.919,Z 627.232,A -85,B 0,C 180,E1 -27085.568,E2 -27085.568} C_VEL
LIN {X 0,Y 90.914,Z 625.951,A -85,B 0,C 180,E1 -27090.001,E2 -27090.001} C_VEL
LIN {X 0,Y 90.971,Z 623.189,A -85,B 0,C 180,E1 -27096.656,E2 -27096.656} C_VEL
LIN {X 0,Y 91.877,Z 619.38,A -85,B 0,C 180,E1 -27103.267,E2 -27103.267} C_VEL
LIN {X 0,Y 93.71,Z 614.419,A -85,B 0,C 180,E1 -27109.725,E2 -27109.725} C_VEL
LIN {X 0,Y 96.65,Z 608.161,A -85,B 0,C 180,E1 -27115.868,E2 -27115.868} C_VEL
LIN {X 0,Y 100.548,Z 600.32,A -85,B 0,C 180,E1 -27121.617,E2 -27121.617} C_VEL
LIN {X 0,Y 103.964,Z 592.977,A -85,B 0,C 180,E1 -27125.786,E2 -27125.786} C_VEL
LIN {X 0,Y 108.317,Z 583.507,A -85,B 0,C 180,E1 -27129.846,E2 -27129.846} C_VEL
LIN {X 0,Y 112.621,Z 572.753,A -85,B 0,C 180,E1 -27133.349,E2 -27133.349} C_VEL
LIN {X 0,Y 116.505,Z 562.424,A -85,B 0,C 180,E1 -27135.753,E2 -27135.753} C_VEL
LIN {X 0,Y 119.812,Z 551.153,A -85,B 0,C 180,E1 -27137.78,E2 -27137.78} C_VEL
LIN {X 0,Y 122.652,Z 538.461,A -85,B 0,C 180,E1 -27139.393,E2 -27139.393} C_VEL
LIN {X 0,Y 124.778,Z 524.93,A -85,B 0,C 180,E1 -27140.492,E2 -27140.492} C_VEL
LIN {X 0,Y 128.112,Z 482.906,A -85,B 0,C 180,E1 -27142.443,E2 -27142.443} C_VEL
LIN {X 0,Y 127.275,Z 480.06,A -85,B 0,C 180,E1 -27143.071,E2 -27143.071} C_VEL
LIN {X 0,Y 125.994,Z 476.925,A -85,B 0,C 180,E1 -27143.961,E2 -27143.961} C_VEL
LIN {X 0,Y 123.376,Z 473.111,A -85,B 0,C 180,E1 -27145.658,E2 -27145.658} C_VEL
LIN {X 0,Y 114.593,Z 464.205,A -85,B 0,C 180,E1 -27152.088,E2 -27152.088} C_VEL
LIN {X 0,Y 113.061,Z 461.755,A -85,B 0,C 180,E1 -27153.539,E2 -27153.539} C_VEL
LIN {X 0,Y 108.819,Z 455.042,A -85,B 0,C 180,E1 -27158.138,E2 -27158.138} C_VEL
LIN {X 0,Y 106.063,Z 451.158,A -85,B 0,C 180,E1 -27161.685,E2 -27161.685} C_VEL
LIN {X 0,Y 104.983,Z 449.843,A -85,B 0,C 180,E1 -27163.22,E2 -27163.22} C_VEL
LIN {X 0,Y 102.821,Z 446.645,A -85,B 0,C 180,E1 -27166.855,E2 -27166.855} C_VEL
LIN {X 0,Y 102.204,Z 445.528,A -85,B 0,C 180,E1 -27168.094,E2 -27168.094} C_VEL
LIN {X 0,Y 99.67,Z 442.74,A -85,B 0,C 180,E1 -27174.055,E2 -27174.055} C_VEL
LIN {X 0,Y 98.838,Z 440.539,A -85,B 0,C 180,E1 -27177.452,E2 -27177.452} C_VEL
LIN {X 0,Y 98.318,Z 439.943,A -85,B 0,C 180,E1 -27180,E2 -27180} C_VEL
LIN {X 0,Y 98.127,Z 440.237,A -85,B 0,C 180,E1 -27192.407,E2 -27192.407} C_VEL
LIN {X 0,Y 98.634,Z 440.965,A -85,B 0,C 180,E1 -27195.241,E2 -27195.241} C_VEL
LIN {X 0,Y 100.069,Z 443.924,A -85,B 0,C 180,E1 -27200.558,E2 -27200.558} C_VEL
LIN {X 0,Y 102.498,Z 446.158,A -85,B 0,C 180,E1 -27205.786,E2 -27205.786} C_VEL
LIN {X 0,Y 104.636,Z 449.602,A -85,B 0,C 180,E1 -27209.551,E2 -27209.551} C_VEL
LIN {X 0,Y 105.911,Z 451.013,A -85,B 0,C 180,E1 -27211.371,E2 -27211.371} C_VEL
LIN {X 0,Y 109.138,Z 455.846,A -85,B 0,C 180,E1 -27215.539,E2 -27215.539} C_VEL
LIN {X 0,Y 113.157,Z 461.97,A -85,B 0,C 180,E1 -27219.817,E2 -27219.817} C_VEL
LIN {X 0,Y 117.632,Z 469.891,A -85,B 0,C 180,E1 -27223.878,E2 -27223.878} C_VEL
LIN {X 0,Y 121.942,Z 478.968,A -85,B 0,C 180,E1 -27227.336,E2 -27227.336} C_VEL
LIN {X 0,Y 123.322,Z 482.151,A -85,B 0,C 180,E1 -27228.368,E2 -27228.368} C_VEL
LIN {X 0,Y 119.96,Z 522.002,A -85,B 0,C 180,E1 -27230.194,E2 -27230.194} C_VEL
LIN {X 0,Y 117.774,Z 535.604,A -85,B 0,C 180,E1 -27231.291,E2 -27231.291} C_VEL
LIN {X 0,Y 114.89,Z 547.962,A -85,B 0,C 180,E1 -27232.839,E2 -27232.839} C_VEL
LIN {X 0,Y 111.332,Z 559.878,A -85,B 0,C 180,E1 -27235.009,E2 -27235.009} C_VEL
LIN {X 0,Y 107.106,Z 571.086,A -85,B 0,C 180,E1 -27237.782,E2 -27237.782} C_VEL
LIN {X 0,Y 102.889,Z 580.564,A -85,B 0,C 180,E1 -27240.877,E2 -27240.877} C_VEL
LIN {X 0,Y 98.682,Z 589.341,A -85,B 0,C 180,E1 -27244.702,E2 -27244.702} C_VEL
LIN {X 0,Y 94.562,Z 597.409,A -85,B 0,C 180,E1 -27249.327,E2 -27249.327} C_VEL
LIN {X 0,Y 90.32,Z 605.334,A -85,B 0,C 180,E1 -27255.351,E2 -27255.351} C_VEL
LIN {X 0,Y 87.665,Z 610.691,A -85,B 0,C 180,E1 -27260.773,E2 -27260.773} C_VEL
LIN {X 0,Y 85.368,Z 615.932,A -85,B 0,C 180,E1 -27267.64,E2 -27267.64} C_VEL
LIN {X 0,Y 83.888,Z 620.018,A -85,B 0,C 180,E1 -27274.804,E2 -27274.804} C_VEL
LIN {X 0,Y 83.33,Z 622.136,A -85,B 0,C 180,E1 -27279.71,E2 -27279.71} C_VEL
LIN {X 0,Y 83.267,Z 623.818,A -85,B 0,C 180,E1 -27284.666,E2 -27284.666} C_VEL
LIN {X 0,Y 84.383,Z 625.802,A -85,B 0,C 180,E1 -27293.63,E2 -27293.63} C_VEL
LIN {X 0,Y 85.901,Z 626.318,A -85,B 0,C 180,E1 -27299.397,E2 -27299.397} C_VEL
LIN {X 0,Y 87.773,Z 626.316,A -85,B 0,C 180,E1 -27304.088,E2 -27304.088} C_VEL
LIN {X 0,Y 90.473,Z 625.827,A -85,B 0,C 180,E1 -27309.031,E2 -27309.031} C_VEL
LIN {X 0,Y 96.456,Z 623.735,A -85,B 0,C 180,E1 -27316.768,E2 -27316.768} C_VEL
LIN {X 0,Y 101.314,Z 621.472,A -85,B 0,C 180,E1 -27321.368,E2 -27321.368} C_VEL
LIN {X 0,Y 108.912,Z 617.077,A -85,B 0,C 180,E1 -27327.018,E2 -27327.018} C_VEL
LIN {X 0,Y 116.855,Z 611.551,A -85,B 0,C 180,E1 -27331.563,E2 -27331.563} C_VEL
LIN {X 0,Y 125.507,Z 604.321,A -85,B 0,C 180,E1 -27335.494,E2 -27335.494} C_VEL
LIN {X 0,Y 133.74,Z 596.138,A -85,B 0,C 180,E1 -27338.562,E2 -27338.562} C_VEL
LIN {X 0,Y 141.232,Z 587.253,A -85,B 0,C 180,E1 -27340.988,E2 -27340.988} C_VEL
LIN {X 0,Y 148.345,Z 577.118,A -85,B 0,C 180,E1 -27342.97,E2 -27342.97} C_VEL
LIN {X 0,Y 154.864,Z 565.69,A -85,B 0,C 180,E1 -27344.651,E2 -27344.651} C_VEL
LIN {X 0,Y 160.168,Z 554.087,A -85,B 0,C 180,E1 -27345.873,E2 -27345.873} C_VEL
LIN {X 0,Y 164.673,Z 541.166,A -85,B 0,C 180,E1 -27346.794,E2 -27346.794} C_VEL
LIN {X 0,Y 167.907,Z 527.881,A -85,B 0,C 180,E1 -27347.462,E2 -27347.462} C_VEL
LIN {X 0,Y 169.058,Z 520.439,A -85,B 0,C 180,E1 -27347.758,E2 -27347.758} C_VEL
LIN {X 0,Y 167.753,Z 516.957,A -85,B 0,C 180,E1 -27349.668,E2 -27349.668} C_VEL
LIN {X 0,Y 165.44,Z 511.891,A -85,B 0,C 180,E1 -27353.445,E2 -27353.445} C_VEL
LIN {X 0,Y 164.238,Z 509.139,A -85,B 0,C 180,E1 -27356.013,E2 -27356.013} C_VEL
LIN {X 0,Y 163.075,Z 506.409,A -85,B 0,C 180,E1 -27359.383,E2 -27359.383} C_VEL
LIN {X 0,Y 162.203,Z 504.691,A -85,B 0,C 180,E1 -27363.727,E2 -27363.727} C_VEL
LIN {X 0,Y 162.055,Z 504.736,A -85,B 0,C 180,E1 -27367.789,E2 -27367.789} C_VEL
LIN {X 0,Y 163.199,Z 507.061,A -85,B 0,C 180,E1 -27374.019,E2 -27374.019} C_VEL
LIN {X 0,Y 164.957,Z 510.922,A -85,B 0,C 180,E1 -27378.474,E2 -27378.474} C_VEL
LIN {X 0,Y 165.872,Z 513.261,A -85,B 0,C 180,E1 -27380.279,E2 -27380.279} C_VEL
LIN {X 0,Y 167.737,Z 518.61,A -85,B 0,C 180,E1 -27383.406,E2 -27383.406} C_VEL
LIN {X 0,Y 168.865,Z 522.522,A -85,B 0,C 180,E1 -27385.185,E2 -27385.185} C_VEL
LIN {X 0,Y 166.717,Z 534.485,A -85,B 0,C 180,E1 -27385.676,E2 -27385.676} C_VEL
LIN {X 0,Y 163.519,Z 546.056,A -85,B 0,C 180,E1 -27386.306,E2 -27386.306} C_VEL
LIN {X 0,Y 158.951,Z 558.2,A -85,B 0,C 180,E1 -27387.251,E2 -27387.251} C_VEL
LIN {X 0,Y 152.955,Z 570.407,A -85,B 0,C 180,E1 -27388.511,E2 -27388.511} C_VEL
LIN {X 0,Y 146.337,Z 581.321,A -85,B 0,C 180,E1 -27390.181,E2 -27390.181} C_VEL
LIN {X 0,Y 139.145,Z 591.089,A -85,B 0,C 180,E1 -27392.222,E2 -27392.222} C_VEL
LIN {X 0,Y 132.179,Z 599.112,A -85,B 0,C 180,E1 -27394.502,E2 -27394.502} C_VEL
LIN {X 0,Y 124.044,Z 607.016,A -85,B 0,C 180,E1 -27397.517,E2 -27397.517} C_VEL
LIN {X 0,Y 116.403,Z 613.355,A -85,B 0,C 180,E1 -27401.003,E2 -27401.003} C_VEL
LIN {X 0,Y 109.419,Z 618.404,A -85,B 0,C 180,E1 -27405.049,E2 -27405.049} C_VEL
LIN {X 0,Y 102.94,Z 622.347,A -85,B 0,C 180,E1 -27409.567,E2 -27409.567} C_VEL
LIN {X 0,Y 97.207,Z 625.275,A -85,B 0,C 180,E1 -27414.664,E2 -27414.664} C_VEL
LIN {X 0,Y 90.844,Z 627.708,A -85,B 0,C 180,E1 -27422.345,E2 -27422.345} C_VEL
LIN {X 0,Y 86.587,Z 628.614,A -85,B 0,C 180,E1 -27431.056,E2 -27431.056} C_VEL
LIN {X 0,Y 85.192,Z 628.478,A -85,B 0,C 180,E1 -27435.673,E2 -27435.673} C_VEL
LIN {X 0,Y 83.859,Z 627.012,A -85,B 0,C 180,E1 -27445.194,E2 -27445.194} C_VEL
LIN {X 0,Y 83.813,Z 625.695,A -85,B 0,C 180,E1 -27450.001,E2 -27450.001} C_VEL
LIN {X 0,Y 83.923,Z 622.861,A -85,B 0,C 180,E1 -27457.217,E2 -27457.217} C_VEL
LIN {X 0,Y 84.964,Z 618.975,A -85,B 0,C 180,E1 -27464.369,E2 -27464.369} C_VEL
LIN {X 0,Y 87.019,Z 613.929,A -85,B 0,C 180,E1 -27471.312,E2 -27471.312} C_VEL
LIN {X 0,Y 90.276,Z 607.574,A -85,B 0,C 180,E1 -27477.847,E2 -27477.847} C_VEL
LIN {X 0,Y 94.564,Z 599.584,A -85,B 0,C 180,E1 -27483.877,E2 -27483.877} C_VEL
LIN {X 0,Y 98.66,Z 591.348,A -85,B 0,C 180,E1 -27488.591,E2 -27488.591} C_VEL
LIN {X 0,Y 103.439,Z 581.405,A -85,B 0,C 180,E1 -27492.8,E2 -27492.8} C_VEL
LIN {X 0,Y 107.561,Z 571.544,A -85,B 0,C 180,E1 -27495.95,E2 -27495.95} C_VEL
LIN {X 0,Y 111.639,Z 560.893,A -85,B 0,C 180,E1 -27498.38,E2 -27498.38} C_VEL
LIN {X 0,Y 115.391,Z 547.961,A -85,B 0,C 180,E1 -27500.601,E2 -27500.601} C_VEL
LIN {X 0,Y 118.302,Z 534.792,A -85,B 0,C 180,E1 -27502.117,E2 -27502.117} C_VEL
LIN {X 0,Y 120.193,Z 521.447,A -85,B 0,C 180,E1 -27503.047,E2 -27503.047} C_VEL
LIN {X 0,Y 123.189,Z 484.942,A -85,B 0,C 180,E1 -27504.715,E2 -27504.715} C_VEL
LIN {X 0,Y 120.383,Z 475.687,A -85,B 0,C 180,E1 -27507.113,E2 -27507.113} C_VEL
LIN {X 0,Y 116.867,Z 468.417,A -85,B 0,C 180,E1 -27510.034,E2 -27510.034} C_VEL
LIN {X 0,Y 113.061,Z 461.755,A -85,B 0,C 180,E1 -27513.539,E2 -27513.539} C_VEL
LIN {X 0,Y 111.569,Z 459.605,A -85,B 0,C 180,E1 -27515.023,E2 -27515.023} C_VEL
LIN {X 0,Y 109.879,Z 458.173,A -85,B 0,C 180,E1 -27516.706,E2 -27516.706} C_VEL
LIN {X 0,Y 106.404,Z 456.641,A -85,B 0,C 180,E1 -27520.442,E2 -27520.442} C_VEL
LIN {X 0,Y 102.582,Z 454.992,A -85,B 0,C 180,E1 -27525.551,E2 -27525.551} C_VEL
LIN {X 0,Y 100.973,Z 452.773,A -85,B 0,C 180,E1 -27528.583,E2 -27528.583} C_VEL
LIN {X 0,Y 100.297,Z 451.902,A -85,B 0,C 180,E1 -27530.038,E2 -27530.038} C_VEL
LIN {X 0,Y 98.224,Z 449.035,A -85,B 0,C 180,E1 -27535.897,E2 -27535.897} C_VEL
LIN {X 0,Y 97.655,Z 447.266,A -85,B 0,C 180,E1 -27538.778,E2 -27538.778} C_VEL
LIN {X 0,Y 96.889,Z 446.99,A -85,B 0,C 180,E1 -27544.159,E2 -27544.159} C_VEL
LIN {X 0,Y 97.45,Z 447.548,A -85,B 0,C 180,E1 -27553.695,E2 -27553.695} C_VEL
LIN {X 0,Y 98.877,Z 450.797,A -85,B 0,C 180,E1 -27559.799,E2 -27559.799} C_VEL
LIN {X 0,Y 100.955,Z 452.967,A -85,B 0,C 180,E1 -27564.688,E2 -27564.688} C_VEL
LIN {X 0,Y 103.134,Z 456.42,A -85,B 0,C 180,E1 -27568.766,E2 -27568.766} C_VEL
LIN {X 0,Y 104.079,Z 457.687,A -85,B 0,C 180,E1 -27570.24,E2 -27570.24} C_VEL
LIN {X 0,Y 106.776,Z 461.942,A -85,B 0,C 180,E1 -27574.015,E2 -27574.015} C_VEL
LIN {X 0,Y 110.246,Z 467.509,A -85,B 0,C 180,E1 -27578.083,E2 -27578.083} C_VEL
LIN {X 0,Y 114.467,Z 475.46,A -85,B 0,C 180,E1 -27582.308,E2 -27582.308} C_VEL
LIN {X 0,Y 118.243,Z 483.931,A -85,B 0,C 180,E1 -27585.651,E2 -27585.651} C_VEL
LIN {X 0,Y 118.536,Z 484.604,A -85,B 0,C 180,E1 -27585.892,E2 -27585.892} C_VEL
LIN {X 0,Y 115.141,Z 522.689,A -85,B 0,C 180,E1 -27587.66,E2 -27587.66} C_VEL
LIN {X 0,Y 112.84,Z 536.194,A -85,B 0,C 180,E1 -27588.768,E2 -27588.768} C_VEL
LIN {X 0,Y 109.917,Z 548.027,A -85,B 0,C 180,E1 -27590.253,E2 -27590.253} C_VEL
LIN {X 0,Y 106.37,Z 559.421,A -85,B 0,C 180,E1 -27592.325,E2 -27592.325} C_VEL
LIN {X 0,Y 101.729,Z 571.163,A -85,B 0,C 180,E1 -27595.252,E2 -27595.252} C_VEL
LIN {X 0,Y 97.267,Z 580.645,A -85,B 0,C 180,E1 -27598.409,E2 -27598.409} C_VEL
LIN {X 0,Y 92.289,Z 590.324,A -85,B 0,C 180,E1 -27602.811,E2 -27602.811} C_VEL
LIN {X 0,Y 87.953,Z 598.242,A -85,B 0,C 180,E1 -27607.693,E2 -27607.693} C_VEL
LIN {X 0,Y 83.45,Z 605.989,A -85,B 0,C 180,E1 -27614.114,E2 -27614.114} C_VEL
LIN {X 0,Y 80.622,Z 611.277,A -85,B 0,C 180,E1 -27619.958,E2 -27619.958} C_VEL
LIN {X 0,Y 78.213,Z 616.402,A -85,B 0,C 180,E1 -27627.424,E2 -27627.424} C_VEL
LIN {X 0,Y 76.694,Z 620.399,A -85,B 0,C 180,E1 -27635.256,E2 -27635.256} C_VEL
LIN {X 0,Y 76.194,Z 622.463,A -85,B 0,C 180,E1 -27640.629,E2 -27640.629} C_VEL
LIN {X 0,Y 76.226,Z 624.105,A -85,B 0,C 180,E1 -27646.056,E2 -27646.056} C_VEL
LIN {X 0,Y 77.468,Z 625.861,A -85,B 0,C 180,E1 -27654.878,E2 -27654.878} C_VEL
LIN {X 0,Y 79.53,Z 626.443,A -85,B 0,C 180,E1 -27662.018,E2 -27662.018} C_VEL
LIN {X 0,Y 81.749,Z 626.4,A -85,B 0,C 180,E1 -27666.996,E2 -27666.996} C_VEL
LIN {X 0,Y 84.506,Z 625.915,A -85,B 0,C 180,E1 -27671.705,E2 -27671.705} C_VEL
LIN {X 0,Y 87.781,Z 624.99,A -85,B 0,C 180,E1 -27676.098,E2 -27676.098} C_VEL
LIN {X 0,Y 91.54,Z 623.652,A -85,B 0,C 180,E1 -27680.149,E2 -27680.149} C_VEL
LIN {X 0,Y 97.698,Z 620.89,A -85,B 0,C 180,E1 -27685.45,E2 -27685.45} C_VEL
LIN {X 0,Y 105.06,Z 616.815,A -85,B 0,C 180,E1 -27690.412,E2 -27690.412} C_VEL
LIN {X 0,Y 113.061,Z 611.508,A -85,B 0,C 180,E1 -27694.623,E2 -27694.623} C_VEL
LIN {X 0,Y 121.196,Z 605.061,A -85,B 0,C 180,E1 -27698.092,E2 -27698.092} C_VEL
LIN {X 0,Y 129.437,Z 597.319,A -85,B 0,C 180,E1 -27700.987,E2 -27700.987} C_VEL
LIN {X 0,Y 137.475,Z 588.287,A -85,B 0,C 180,E1 -27703.436,E2 -27703.436} C_VEL
LIN {X 0,Y 144.433,Z 578.972,A -85,B 0,C 180,E1 -27705.255,E2 -27705.255} C_VEL
LIN {X 0,Y 150.901,Z 568.394,A -85,B 0,C 180,E1 -27706.808,E2 -27706.808} C_VEL
LIN {X 0,Y 156.284,Z 557.563,A -85,B 0,C 180,E1 -27707.974,E2 -27707.974} C_VEL
LIN {X 0,Y 160.902,Z 545.818,A -85,B 0,C 180,E1 -27708.869,E2 -27708.869} C_VEL
LIN {X 0,Y 164.61,Z 532.971,A -85,B 0,C 180,E1 -27709.555,E2 -27709.555} C_VEL
LIN {X 0,Y 166.313,Z 524.362,A -85,B 0,C 180,E1 -27709.888,E2 -27709.888} C_VEL
LIN {X 0,Y 164.382,Z 519.206,A -85,B 0,C 180,E1 -27713.556,E2 -27713.556} C_VEL
LIN {X 0,Y 163.013,Z 515.814,A -85,B 0,C 180,E1 -27716.756,E2 -27716.756} C_VEL
LIN {X 0,Y 162.094,Z 513.386,A -85,B 0,C 180,E1 -27719.69,E2 -27719.69} C_VEL
LIN {X 0,Y 161.322,Z 511.748,A -85,B 0,C 180,E1 -27723.747,E2 -27723.747} C_VEL
LIN {X 0,Y 161.165,Z 511.743,A -85,B 0,C 180,E1 -27727.517,E2 -27727.517} C_VEL
LIN {X 0,Y 162.135,Z 513.932,A -85,B 0,C 180,E1 -27733.473,E2 -27733.473} C_VEL
LIN {X 0,Y 163.769,Z 517.842,A -85,B 0,C 180,E1 -27737.966,E2 -27737.966} C_VEL
LIN {X 0,Y 164.617,Z 520.537,A -85,B 0,C 180,E1 -27739.903,E2 -27739.903} C_VEL
LIN {X 0,Y 166.061,Z 525.855,A -85,B 0,C 180,E1 -27742.907,E2 -27742.907} C_VEL
LIN {X 0,Y 165.998,Z 526.96,A -85,B 0,C 180,E1 -27743.088,E2 -27743.088} C_VEL
LIN {X 0,Y 163.181,Z 539.391,A -85,B 0,C 180,E1 -27743.578,E2 -27743.578} C_VEL
LIN {X 0,Y 159.377,Z 551.128,A -85,B 0,C 180,E1 -27744.277,E2 -27744.277} C_VEL
LIN {X 0,Y 154.409,Z 562.667,A -85,B 0,C 180,E1 -27745.232,E2 -27745.232} C_VEL
LIN {X 0,Y 148.201,Z 574.02,A -85,B 0,C 180,E1 -27746.484,E2 -27746.484} C_VEL
LIN {X 0,Y 141.442,Z 584.243,A -85,B 0,C 180,E1 -27748.124,E2 -27748.124} C_VEL
LIN {X 0,Y 134.071,Z 593.455,A -85,B 0,C 180,E1 -27750.129,E2 -27750.129} C_VEL
LIN {X 0,Y 125.466,Z 602.404,A -85,B 0,C 180,E1 -27752.839,E2 -27752.839} C_VEL
LIN {X 0,Y 117.17,Z 609.634,A -85,B 0,C 180,E1 -27755.932,E2 -27755.932} C_VEL
LIN {X 0,Y 109.355,Z 615.438,A -85,B 0,C 180,E1 -27759.54,E2 -27759.54} C_VEL
LIN {X 0,Y 103.125,Z 619.438,A -85,B 0,C 180,E1 -27763.145,E2 -27763.145} C_VEL
LIN {X 0,Y 95.475,Z 623.537,A -85,B 0,C 180,E1 -27768.512,E2 -27768.512} C_VEL
LIN {X 0,Y 91.485,Z 625.343,A -85,B 0,C 180,E1 -27772.082,E2 -27772.082} C_VEL
LIN {X 0,Y 84.606,Z 627.693,A -85,B 0,C 180,E1 -27780.107,E2 -27780.107} C_VEL
LIN {X 0,Y 79.872,Z 628.521,A -85,B 0,C 180,E1 -27789.394,E2 -27789.394} C_VEL
LIN {X 0,Y 77.282,Z 627.749,A -85,B 0,C 180,E1 -27799.522,E2 -27799.522} C_VEL
LIN {X 0,Y 76.786,Z 626.792,A -85,B 0,C 180,E1 -27804.75,E2 -27804.75} C_VEL
LIN {X 0,Y 76.734,Z 625.439,A -85,B 0,C 180,E1 -27810.001,E2 -27810.001} C_VEL
LIN {X 0,Y 76.877,Z 622.533,A -85,B 0,C 180,E1 -27817.883,E2 -27817.883} C_VEL
LIN {X 0,Y 78.066,Z 618.568,A -85,B 0,C 180,E1 -27825.67,E2 -27825.67} C_VEL
LIN {X 0,Y 80.913,Z 612.432,A -85,B 0,C 180,E1 -27834.368,E2 -27834.368} C_VEL
LIN {X 0,Y 84.761,Z 605.71,A -85,B 0,C 180,E1 -27841.214,E2 -27841.214} C_VEL
LIN {X 0,Y 89.592,Z 597.341,A -85,B 0,C 180,E1 -27847.441,E2 -27847.441} C_VEL
LIN {X 0,Y 92.91,Z 590.983,A -85,B 0,C 180,E1 -27851.079,E2 -27851.079} C_VEL
LIN {X 0,Y 98.288,Z 580.361,A -85,B 0,C 180,E1 -27855.647,E2 -27855.647} C_VEL
LIN {X 0,Y 102.141,Z 571.645,A -85,B 0,C 180,E1 -27858.441,E2 -27858.441} C_VEL
LIN {X 0,Y 106.41,Z 561.057,A -85,B 0,C 180,E1 -27860.9,E2 -27860.9} C_VEL
LIN {X 0,Y 110.357,Z 548.2,A -85,B 0,C 180,E1 -27863.133,E2 -27863.133} C_VEL
LIN {X 0,Y 113.378,Z 535.257,A -85,B 0,C 180,E1 -27864.651,E2 -27864.651} C_VEL
LIN {X 0,Y 115.299,Z 522.891,A -85,B 0,C 180,E1 -27865.548,E2 -27865.548} C_VEL
LIN {X 0,Y 118.427,Z 486.695,A -85,B 0,C 180,E1 -27867.229,E2 -27867.229} C_VEL
LIN {X 0,Y 116.242,Z 479.309,A -85,B 0,C 180,E1 -27869.33,E2 -27869.33} C_VEL
LIN {X 0,Y 113.167,Z 472.915,A -85,B 0,C 180,E1 -27872.177,E2 -27872.177} C_VEL
LIN {X 0,Y 109.271,Z 465.851,A -85,B 0,C 180,E1 -27876.251,E2 -27876.251} C_VEL
LIN {X 0,Y 106.111,Z 460.72,A -85,B 0,C 180,E1 -27880.141,E2 -27880.141} C_VEL
LIN {X 0,Y 103.33,Z 456.481,A -85,B 0,C 180,E1 -27884.213,E2 -27884.213} C_VEL
LIN {X 0,Y 101.201,Z 453.3,A -85,B 0,C 180,E1 -27888.07,E2 -27888.07} C_VEL
LIN {X 0,Y 100.973,Z 452.773,A -85,B 0,C 180,E1 -27888.583,E2 -27888.583} C_VEL
LIN {X 0,Y 100.095,Z 451.344,A -85,B 0,C 180,E1 -27890.58,E2 -27890.58} C_VEL
LIN {X 0,Y 99.175,Z 450.778,A -85,B 0,C 180,E1 -27892.741,E2 -27892.741} C_VEL
LIN {X 0,Y 98.297,Z 450.856,A -85,B 0,C 180,E1 -27894.996,E2 -27894.996} C_VEL
LIN {X 0,Y 95.947,Z 453.989,A -85,B 0,C 180,E1 -27905.759,E2 -27905.759} C_VEL
LIN {X 0,Y 95.922,Z 454.09,A -85,B 0,C 180,E1 -27907.004,E2 -27907.004} C_VEL
LIN {X 0,Y 96.469,Z 454.649,A -85,B 0,C 180,E1 -27913.23,E2 -27913.23} C_VEL
LIN {X 0,Y 97.703,Z 457.67,A -85,B 0,C 180,E1 -27919.022,E2 -27919.022} C_VEL
LIN {X 0,Y 99.391,Z 459.583,A -85,B 0,C 180,E1 -27923.393,E2 -27923.393} C_VEL
LIN {X 0,Y 102.239,Z 464.27,A -85,B 0,C 180,E1 -27928.984,E2 -27928.984} C_VEL
LIN {X 0,Y 104.769,Z 468.483,A -85,B 0,C 180,E1 -27932.821,E2 -27932.821} C_VEL
LIN {X 0,Y 107.783,Z 473.712,A -85,B 0,C 180,E1 -27936.669,E2 -27936.669} C_VEL
LIN {X 0,Y 111.189,Z 480.624,A -85,B 0,C 180,E1 -27940.444,E2 -27940.444} C_VEL
LIN {X 0,Y 113.947,Z 487.146,A -85,B 0,C 180,E1 -27943.195,E2 -27943.195} C_VEL
LIN {X 0,Y 112.381,Z 505.838,A -85,B 0,C 180,E1 -27944.101,E2 -27944.101} C_VEL
LIN {X 0,Y 110.306,Z 524.921,A -85,B 0,C 180,E1 -27944.991,E2 -27944.991} C_VEL
LIN {X 0,Y 107.883,Z 537.953,A -85,B 0,C 180,E1 -27946.133,E2 -27946.133} C_VEL
LIN {X 0,Y 105.137,Z 548.327,A -85,B 0,C 180,E1 -27947.473,E2 -27947.473} C_VEL
LIN {X 0,Y 101.661,Z 558.977,A -85,B 0,C 180,E1 -27949.405,E2 -27949.405} C_VEL
LIN {X 0,Y 97.197,Z 569.937,A -85,B 0,C 180,E1 -27952.076,E2 -27952.076} C_VEL
LIN {X 0,Y 92.373,Z 579.659,A -85,B 0,C 180,E1 -27955.206,E2 -27955.206} C_VEL
LIN {X 0,Y 88.12,Z 587.713,A -85,B 0,C 180,E1 -27958.774,E2 -27958.774} C_VEL
LIN {X 0,Y 83.193,Z 596.09,A -85,B 0,C 180,E1 -27963.671,E2 -27963.671} C_VEL
LIN {X 0,Y 78.114,Z 604.286,A -85,B 0,C 180,E1 -27970.281,E2 -27970.281} C_VEL
LIN {X 0,Y 74.738,Z 609.86,A -85,B 0,C 180,E1 -27976.402,E2 -27976.402} C_VEL
LIN {X 0,Y 71.771,Z 615.308,A -85,B 0,C 180,E1 -27984.379,E2 -27984.379} C_VEL
LIN {X 0,Y 69.907,Z 619.579,A -85,B 0,C 180,E1 -27992.877,E2 -27992.877} C_VEL
LIN {X 0,Y 69.048,Z 622.792,A -85,B 0,C 180,E1 -28001.744,E2 -28001.744} C_VEL
LIN {X 0,Y 69.246,Z 624.392,A -85,B 0,C 180,E1 -28007.725,E2 -28007.725} C_VEL
LIN {X 0,Y 70.58,Z 625.916,A -85,B 0,C 180,E1 -28016.341,E2 -28016.341} C_VEL
LIN {X 0,Y 73.345,Z 626.569,A -85,B 0,C 180,E1 -28025.092,E2 -28025.092} C_VEL
LIN {X 0,Y 78.255,Z 626.115,A -85,B 0,C 180,E1 -28034.072,E2 -28034.072} C_VEL
LIN {X 0,Y 82.801,Z 624.95,A -85,B 0,C 180,E1 -28039.807,E2 -28039.807} C_VEL
LIN {X 0,Y 86.966,Z 623.569,A -85,B 0,C 180,E1 -28043.91,E2 -28043.91} C_VEL
LIN {X 0,Y 93.931,Z 620.611,A -85,B 0,C 180,E1 -28049.362,E2 -28049.362} C_VEL
LIN {X 0,Y 101.608,Z 616.551,A -85,B 0,C 180,E1 -28054.045,E2 -28054.045} C_VEL
LIN {X 0,Y 111.166,Z 610.321,A -85,B 0,C 180,E1 -28058.573,E2 -28058.573} C_VEL
LIN {X 0,Y 120.139,Z 603.266,A -85,B 0,C 180,E1 -28061.91,E2 -28061.91} C_VEL
LIN {X 0,Y 128.13,Z 595.769,A -85,B 0,C 180,E1 -28064.386,E2 -28064.386} C_VEL
LIN {X 0,Y 135.57,Z 587.477,A -85,B 0,C 180,E1 -28066.403,E2 -28066.403} C_VEL
LIN {X 0,Y 143.554,Z 576.71,A -85,B 0,C 180,E1 -28068.268,E2 -28068.268} C_VEL
LIN {X 0,Y 150.016,Z 565.958,A -85,B 0,C 180,E1 -28069.667,E2 -28069.667} C_VEL
LIN {X 0,Y 155.75,Z 554.017,A -85,B 0,C 180,E1 -28070.769,E2 -28070.769} C_VEL
LIN {X 0,Y 160.283,Z 541.566,A -85,B 0,C 180,E1 -28071.554,E2 -28071.554} C_VEL
LIN {X 0,Y 163.515,Z 529.102,A -85,B 0,C 180,E1 -28072.108,E2 -28072.108} C_VEL
LIN {X 0,Y 163.604,Z 528.584,A -85,B 0,C 180,E1 -28072.163,E2 -28072.163} C_VEL
LIN {X 0,Y 161.956,Z 523.106,A -85,B 0,C 180,E1 -28076.701,E2 -28076.701} C_VEL
LIN {X 0,Y 160.963,Z 520.216,A -85,B 0,C 180,E1 -28080.337,E2 -28080.337} C_VEL
LIN {X 0,Y 160.412,Z 518.8,A -85,B 0,C 180,E1 -28083.768,E2 -28083.768} C_VEL
LIN {X 0,Y 160.236,Z 518.703,A -85,B 0,C 180,E1 -28086.295,E2 -28086.295} C_VEL
LIN {X 0,Y 160.601,Z 520.031,A -85,B 0,C 180,E1 -28091.038,E2 -28091.038} C_VEL
LIN {X 0,Y 161.054,Z 520.92,A -85,B 0,C 180,E1 -28093.084,E2 -28093.084} C_VEL
LIN {X 0,Y 162.284,Z 524.394,A -85,B 0,C 180,E1 -28097.159,E2 -28097.159} C_VEL
LIN {X 0,Y 163.17,Z 528.149,A -85,B 0,C 180,E1 -28099.8,E2 -28099.8} C_VEL
LIN {X 0,Y 163.489,Z 529.808,A -85,B 0,C 180,E1 -28100.757,E2 -28100.757} C_VEL
LIN {X 0,Y 160.337,Z 542.214,A -85,B 0,C 180,E1 -28101.321,E2 -28101.321} C_VEL
LIN {X 0,Y 156.064,Z 554.139,A -85,B 0,C 180,E1 -28102.044,E2 -28102.044} C_VEL
LIN {X 0,Y 150.748,Z 565.491,A -85,B 0,C 180,E1 -28102.967,E2 -28102.967} C_VEL
LIN {X 0,Y 144.424,Z 576.23,A -85,B 0,C 180,E1 -28104.163,E2 -28104.163} C_VEL
LIN {X 0,Y 136.724,Z 586.938,A -85,B 0,C 180,E1 -28105.905,E2 -28105.905} C_VEL
LIN {X 0,Y 129.171,Z 595.66,A -85,B 0,C 180,E1 -28107.858,E2 -28107.858} C_VEL
LIN {X 0,Y 120.315,Z 604.189,A -85,B 0,C 180,E1 -28110.507,E2 -28110.507} C_VEL
LIN {X 0,Y 111.762,Z 611.024,A -85,B 0,C 180,E1 -28113.574,E2 -28113.574} C_VEL
LIN {X 0,Y 102.394,Z 617.315,A -85,B 0,C 180,E1 -28117.881,E2 -28117.881} C_VEL
LIN {X 0,Y 94.972,Z 621.453,A -85,B 0,C 180,E1 -28122.271,E2 -28122.271} C_VEL
LIN {X 0,Y 90.282,Z 623.661,A -85,B 0,C 180,E1 -28125.527,E2 -28125.527} C_VEL
LIN {X 0,Y 82.039,Z 626.73,A -85,B 0,C 180,E1 -28133.157,E2 -28133.157} C_VEL
LIN {X 0,Y 75.581,Z 628.249,A -85,B 0,C 180,E1 -28142.296,E2 -28142.296} C_VEL
LIN {X 0,Y 71.483,Z 628.174,A -85,B 0,C 180,E1 -28152.847,E2 -28152.847} C_VEL
LIN {X 0,Y 69.734,Z 626.572,A -85,B 0,C 180,E1 -28164.217,E2 -28164.217} C_VEL
LIN {X 0,Y 69.646,Z 625.162,A -85,B 0,C 180,E1 -28170.001,E2 -28170.001} C_VEL
LIN {X 0,Y 69.826,Z 622.193,A -85,B 0,C 180,E1 -28178.685,E2 -28178.685} C_VEL
LIN {X 0,Y 71.23,Z 618.151,A -85,B 0,C 180,E1 -28187.219,E2 -28187.219} C_VEL
LIN {X 0,Y 74.469,Z 611.899,A -85,B 0,C 180,E1 -28196.634,E2 -28196.634} C_VEL
LIN {X 0,Y 78.742,Z 605.08,A -85,B 0,C 180,E1 -28203.907,E2 -28203.907} C_VEL
LIN {X 0,Y 83.967,Z 596.559,A -85,B 0,C 180,E1 -28210.442,E2 -28210.442} C_VEL
LIN {X 0,Y 87.918,Z 589.663,A -85,B 0,C 180,E1 -28214.382,E2 -28214.382} C_VEL
LIN {X 0,Y 92.851,Z 580.432,A -85,B 0,C 180,E1 -28218.37,E2 -28218.37} C_VEL
LIN {X 0,Y 96.935,Z 571.741,A -85,B 0,C 180,E1 -28221.206,E2 -28221.206} C_VEL
LIN {X 0,Y 101.41,Z 561.216,A -85,B 0,C 180,E1 -28223.672,E2 -28223.672} C_VEL
LIN {X 0,Y 105.244,Z 549.587,A -85,B 0,C 180,E1 -28225.729,E2 -28225.729} C_VEL
LIN {X 0,Y 108.533,Z 536.436,A -85,B 0,C 180,E1 -28227.331,E2 -28227.331} C_VEL
LIN {X 0,Y 110.727,Z 523.645,A -85,B 0,C 180,E1 -28228.293,E2 -28228.293} C_VEL
LIN {X 0,Y 113.974,Z 488.806,A -85,B 0,C 180,E1 -28229.866,E2 -28229.866} C_VEL
LIN {X 0,Y 112.291,Z 483.184,A -85,B 0,C 180,E1 -28231.678,E2 -28231.678} C_VEL
LIN {X 0,Y 109.788,Z 477.63,A -85,B 0,C 180,E1 -28234.305,E2 -28234.305} C_VEL
LIN {X 0,Y 106.406,Z 471.143,A -85,B 0,C 180,E1 -28238.285,E2 -28238.285} C_VEL
LIN {X 0,Y 103.759,Z 466.665,A -85,B 0,C 180,E1 -28241.903,E2 -28241.903} C_VEL
LIN {X 0,Y 101.493,Z 462.927,A -85,B 0,C 180,E1 -28245.593,E2 -28245.593} C_VEL
LIN {X 0,Y 99.357,Z 459.253,A -85,B 0,C 180,E1 -28250.013,E2 -28250.013} C_VEL
LIN {X 0,Y 96.974,Z 455.585,A -85,B 0,C 180,E1 -28257.328,E2 -28257.328} C_VEL
LIN {X 0,Y 96.542,Z 454.097,A -85,B 0,C 180,E1 -28260,E2 -28260} C_VEL
LIN {X 0,Y 95.922,Z 454.09,A -85,B 0,C 180,E1 -28267.004,E2 -28267.004} C_VEL
LIN {X 0,Y 95.965,Z 454.577,A -85,B 0,C 180,E1 -28269.317,E2 -28269.317} C_VEL
LIN {X 0,Y 96.133,Z 456.545,A -85,B 0,C 180,E1 -28272.63,E2 -28272.63} C_VEL
LIN {X 0,Y 96.447,Z 459.417,A -85,B 0,C 180,E1 -28275.724,E2 -28275.724} C_VEL
LIN {X 0,Y 97.793,Z 465.923,A -85,B 0,C 180,E1 -28281.794,E2 -28281.794} C_VEL
LIN {X 0,Y 98.588,Z 467.707,A -85,B 0,C 180,E1 -28283.876,E2 -28283.876} C_VEL
LIN {X 0,Y 100.296,Z 470.5,A -85,B 0,C 180,E1 -28287.38,E2 -28287.38} C_VEL
LIN {X 0,Y 102.793,Z 475.045,A -85,B 0,C 180,E1 -28291.575,E2 -28291.575} C_VEL
LIN {X 0,Y 105.389,Z 479.922,A -85,B 0,C 180,E1 -28295.192,E2 -28295.192} C_VEL
LIN {X 0,Y 108.295,Z 486.315,A -85,B 0,C 180,E1 -28298.76,E2 -28298.76} C_VEL
LIN {X 0,Y 109.724,Z 489.87,A -85,B 0,C 180,E1 -28300.373,E2 -28300.373} C_VEL
LIN {X 0,Y 106.485,Z 522.688,A -85,B 0,C 180,E1 -28301.851,E2 -28301.851} C_VEL
LIN {X 0,Y 103.972,Z 536.257,A -85,B 0,C 180,E1 -28302.918,E2 -28302.918} C_VEL
LIN {X 0,Y 100.708,Z 548.347,A -85,B 0,C 180,E1 -28304.394,E2 -28304.394} C_VEL
LIN {X 0,Y 97.1,Z 558.87,A -85,B 0,C 180,E1 -28306.273,E2 -28306.273} C_VEL
LIN {X 0,Y 92.329,Z 570.014,A -85,B 0,C 180,E1 -28308.964,E2 -28308.964} C_VEL
LIN {X 0,Y 87.231,Z 579.74,A -85,B 0,C 180,E1 -28312.096,E2 -28312.096} C_VEL
LIN {X 0,Y 82.115,Z 588.695,A -85,B 0,C 180,E1 -28316.198,E2 -28316.198} C_VEL
LIN {X 0,Y 76.882,Z 596.925,A -85,B 0,C 180,E1 -28321.319,E2 -28321.319} C_VEL
LIN {X 0,Y 71.452,Z 604.996,A -85,B 0,C 180,E1 -28328.354,E2 -28328.354} C_VEL
LIN {X 0,Y 67.826,Z 610.46,A -85,B 0,C 180,E1 -28334.985,E2 -28334.985} C_VEL
LIN {X 0,Y 64.678,Z 615.809,A -85,B 0,C 180,E1 -28343.76,E2 -28343.76} C_VEL
LIN {X 0,Y 62.706,Z 619.992,A -85,B 0,C 180,E1 -28353.208,E2 -28353.208} C_VEL
LIN {X 0,Y 61.952,Z 623.121,A -85,B 0,C 180,E1 -28363.112,E2 -28363.112} C_VEL
LIN {X 0,Y 62.315,Z 624.662,A -85,B 0,C 180,E1 -28369.774,E2 -28369.774} C_VEL
LIN {X 0,Y 63.756,Z 625.973,A -85,B 0,C 180,E1 -28378.133,E2 -28378.133} C_VEL
LIN {X 0,Y 67.406,Z 626.694,A -85,B 0,C 180,E1 -28388.722,E2 -28388.722} C_VEL
LIN {X 0,Y 72.409,Z 626.251,A -85,B 0,C 180,E1 -28397.202,E2 -28397.202} C_VEL
LIN {X 0,Y 78.217,Z 624.909,A -85,B 0,C 180,E1 -28403.963,E2 -28403.963} C_VEL
LIN {X 0,Y 86.452,Z 622.101,A -85,B 0,C 180,E1 -28410.807,E2 -28410.807} C_VEL
LIN {X 0,Y 95.779,Z 617.754,A -85,B 0,C 180,E1 -28416.518,E2 -28416.518} C_VEL
LIN {X 0,Y 104.38,Z 612.786,A -85,B 0,C 180,E1 -28420.493,E2 -28420.493} C_VEL
LIN {X 0,Y 113.414,Z 606.478,A -85,B 0,C 180,E1 -28423.836,E2 -28423.836} C_VEL
LIN {X 0,Y 122.794,Z 598.56,A -85,B 0,C 180,E1 -28426.643,E2 -28426.643} C_VEL
LIN {X 0,Y 130.783,Z 590.38,A -85,B 0,C 180,E1 -28428.719,E2 -28428.719} C_VEL
LIN {X 0,Y 138.947,Z 580.361,A -85,B 0,C 180,E1 -28430.5,E2 -28430.5} C_VEL
LIN {X 0,Y 146.122,Z 569.526,A -85,B 0,C 180,E1 -28431.937,E2 -28431.937} C_VEL
LIN {X 0,Y 152.226,Z 557.94,A -85,B 0,C 180,E1 -28433.018,E2 -28433.018} C_VEL
LIN {X 0,Y 157.057,Z 546.2,A -85,B 0,C 180,E1 -28433.795,E2 -28433.795} C_VEL
LIN {X 0,Y 160.988,Z 533.115,A -85,B 0,C 180,E1 -28434.412,E2 -28434.412} C_VEL
LIN {X 0,Y 160.087,Z 529.148,A -85,B 0,C 180,E1 -28438.113,E2 -28438.113} C_VEL
LIN {X 0,Y 159.578,Z 527.015,A -85,B 0,C 180,E1 -28440.947,E2 -28440.947} C_VEL
LIN {X 0,Y 159.18,Z 525.712,A -85,B 0,C 180,E1 -28444.432,E2 -28444.432} C_VEL
LIN {X 0,Y 159.077,Z 525.951,A -85,B 0,C 180,E1 -28447.617,E2 -28447.617} C_VEL
LIN {X 0,Y 159.66,Z 527.732,A -85,B 0,C 180,E1 -28452.553,E2 -28452.553} C_VEL
LIN {X 0,Y 160.594,Z 531.275,A -85,B 0,C 180,E1 -28456.745,E2 -28456.745} C_VEL
LIN {X 0,Y 160.926,Z 533.96,A -85,B 0,C 180,E1 -28458.491,E2 -28458.491} C_VEL
LIN {X 0,Y 157.188,Z 546.542,A -85,B 0,C 180,E1 -28459.054,E2 -28459.054} C_VEL
LIN {X 0,Y 152.108,Z 558.937,A -85,B 0,C 180,E1 -28459.835,E2 -28459.835} C_VEL
LIN {X 0,Y 145.704,Z 570.938,A -85,B 0,C 180,E1 -28460.849,E2 -28460.849} C_VEL
LIN {X 0,Y 138.523,Z 581.661,A -85,B 0,C 180,E1 -28462.198,E2 -28462.198} C_VEL
LIN {X 0,Y 130.649,Z 591.321,A -85,B 0,C 180,E1 -28463.872,E2 -28463.872} C_VEL
LIN {X 0,Y 122.975,Z 599.244,A -85,B 0,C 180,E1 -28465.832,E2 -28465.832} C_VEL
LIN {X 0,Y 113.908,Z 607.054,A -85,B 0,C 180,E1 -28468.457,E2 -28468.457} C_VEL
LIN {X 0,Y 106.556,Z 612.358,A -85,B 0,C 180,E1 -28470.975,E2 -28470.975} C_VEL
LIN {X 0,Y 98.197,Z 617.558,A -85,B 0,C 180,E1 -28474.611,E2 -28474.611} C_VEL
LIN {X 0,Y 90.344,Z 621.618,A -85,B 0,C 180,E1 -28478.933,E2 -28478.933} C_VEL
LIN {X 0,Y 85.366,Z 623.762,A -85,B 0,C 180,E1 -28482.191,E2 -28482.191} C_VEL
LIN {X 0,Y 76.471,Z 626.749,A -85,B 0,C 180,E1 -28489.962,E2 -28489.962} C_VEL
LIN {X 0,Y 69.346,Z 628.183,A -85,B 0,C 180,E1 -28499.556,E2 -28499.556} C_VEL
LIN {X 0,Y 64.727,Z 628.022,A -85,B 0,C 180,E1 -28510.992,E2 -28510.992} C_VEL
LIN {X 0,Y 62.664,Z 626.348,A -85,B 0,C 180,E1 -28523.562,E2 -28523.562} C_VEL
LIN {X 0,Y 62.547,Z 624.871,A -85,B 0,C 180,E1 -28530.002,E2 -28530.002} C_VEL
LIN {X 0,Y 62.808,Z 621.831,A -85,B 0,C 180,E1 -28539.664,E2 -28539.664} C_VEL
LIN {X 0,Y 64.464,Z 617.71,A -85,B 0,C 180,E1 -28549.092,E2 -28549.092} C_VEL
LIN {X 0,Y 68.17,Z 611.366,A -85,B 0,C 180,E1 -28559.322,E2 -28559.322} C_VEL
LIN {X 0,Y 72.91,Z 604.449,A -85,B 0,C 180,E1 -28567.047,E2 -28567.047} C_VEL
LIN {X 0,Y 78.337,Z 596.206,A -85,B 0,C 180,E1 -28573.561,E2 -28573.561} C_VEL
LIN {X 0,Y 84.116,Z 586.806,A -85,B 0,C 180,E1 -28578.761,E2 -28578.761} C_VEL
LIN {X 0,Y 89.443,Z 576.943,A -85,B 0,C 180,E1 -28582.71,E2 -28582.71} C_VEL
LIN {X 0,Y 94.611,Z 566.14,A -85,B 0,C 180,E1 -28585.731,E2 -28585.731} C_VEL
LIN {X 0,Y 98.992,Z 554.989,A -85,B 0,C 180,E1 -28587.942,E2 -28587.942} C_VEL
LIN {X 0,Y 102.766,Z 542.57,A -85,B 0,C 180,E1 -28589.701,E2 -28589.701} C_VEL
LIN {X 0,Y 105.539,Z 530.118,A -85,B 0,C 180,E1 -28590.857,E2 -28590.857} C_VEL
LIN {X 0,Y 107.272,Z 516.763,A -85,B 0,C 180,E1 -28591.643,E2 -28591.643} C_VEL
LIN {X 0,Y 109.725,Z 490.768,A -85,B 0,C 180,E1 -28592.774,E2 -28592.774} C_VEL
LIN {X 0,Y 108.295,Z 486.224,A -85,B 0,C 180,E1 -28594.506,E2 -28594.506} C_VEL
LIN {X 0,Y 104.712,Z 478.461,A -85,B 0,C 180,E1 -28598.982,E2 -28598.982} C_VEL
LIN {X 0,Y 101.869,Z 473.103,A -85,B 0,C 180,E1 -28603.175,E2 -28603.175} C_VEL
LIN {X 0,Y 99.601,Z 469.157,A -85,B 0,C 180,E1 -28607.261,E2 -28607.261} C_VEL
LIN {X 0,Y 97.582,Z 465.406,A -85,B 0,C 180,E1 -28612.081,E2 -28612.081} C_VEL
LIN {X 0,Y 95.862,Z 462.424,A -85,B 0,C 180,E1 -28618.311,E2 -28618.311} C_VEL
LIN {X 0,Y 95.55,Z 461.13,A -85,B 0,C 180,E1 -28620.621,E2 -28620.621} C_VEL
LIN {X 0,Y 95.375,Z 461.351,A -85,B 0,C 180,E1 -28631.691,E2 -28631.691} C_VEL
LIN {X 0,Y 97.055,Z 465.204,A -85,B 0,C 180,E1 -28639.841,E2 -28639.841} C_VEL
LIN {X 0,Y 97.938,Z 466.313,A -85,B 0,C 180,E1 -28642.215,E2 -28642.215} C_VEL
LIN {X 0,Y 98.588,Z 467.707,A -85,B 0,C 180,E1 -28643.876,E2 -28643.876} C_VEL
LIN {X 0,Y 99.864,Z 470.663,A -85,B 0,C 180,E1 -28646.741,E2 -28646.741} C_VEL
LIN {X 0,Y 101.023,Z 474.58,A -85,B 0,C 180,E1 -28649.211,E2 -28649.211} C_VEL
LIN {X 0,Y 103.161,Z 483.887,A -85,B 0,C 180,E1 -28653.41,E2 -28653.41} C_VEL
LIN {X 0,Y 104.807,Z 490.244,A -85,B 0,C 180,E1 -28656.073,E2 -28656.073} C_VEL
LIN {X 0,Y 105.727,Z 492.694,A -85,B 0,C 180,E1 -28657.291,E2 -28657.291} C_VEL
LIN {X 0,Y 102.518,Z 523.265,A -85,B 0,C 180,E1 -28658.625,E2 -28658.625} C_VEL
LIN {X 0,Y 99.852,Z 536.897,A -85,B 0,C 180,E1 -28659.679,E2 -28659.679} C_VEL
LIN {X 0,Y 96.248,Z 549.461,A -85,B 0,C 180,E1 -28661.198,E2 -28661.198} C_VEL
LIN {X 0,Y 92.096,Z 560.604,A -85,B 0,C 180,E1 -28663.216,E2 -28663.216} C_VEL
LIN {X 0,Y 87.069,Z 571.395,A -85,B 0,C 180,E1 -28665.878,E2 -28665.878} C_VEL
LIN {X 0,Y 81.773,Z 580.89,A -85,B 0,C 180,E1 -28669.055,E2 -28669.055} C_VEL
LIN {X 0,Y 76.278,Z 589.681,A -85,B 0,C 180,E1 -28673.209,E2 -28673.209} C_VEL
LIN {X 0,Y 70.728,Z 597.759,A -85,B 0,C 180,E1 -28678.554,E2 -28678.554} C_VEL
LIN {X 0,Y 64.861,Z 605.695,A -85,B 0,C 180,E1 -28686.024,E2 -28686.024} C_VEL
LIN {X 0,Y 60.965,Z 611.06,A -85,B 0,C 180,E1 -28693.248,E2 -28693.248} C_VEL
LIN {X 0,Y 57.564,Z 616.31,A -85,B 0,C 180,E1 -28702.986,E2 -28702.986} C_VEL
LIN {X 0,Y 55.479,Z 620.406,A -85,B 0,C 180,E1 -28713.63,E2 -28713.63} C_VEL
LIN {X 0,Y 54.865,Z 623.45,A -85,B 0,C 180,E1 -28724.842,E2 -28724.842} C_VEL
LIN {X 0,Y 55.486,Z 624.909,A -85,B 0,C 180,E1 -28732.331,E2 -28732.331} C_VEL
LIN {X 0,Y 57.016,Z 626.031,A -85,B 0,C 180,E1 -28740.363,E2 -28740.363} C_VEL
LIN {X 0,Y 61.789,Z 626.8,A -85,B 0,C 180,E1 -28753.032,E2 -28753.032} C_VEL
LIN {X 0,Y 66.874,Z 626.377,A -85,B 0,C 180,E1 -28760.91,E2 -28760.91} C_VEL
LIN {X 0,Y 74.089,Z 624.87,A -85,B 0,C 180,E1 -28768.616,E2 -28768.616} C_VEL
LIN {X 0,Y 82.077,Z 622.33,A -85,B 0,C 180,E1 -28774.651,E2 -28774.651} C_VEL
LIN {X 0,Y 90.159,Z 618.943,A -85,B 0,C 180,E1 -28779.29,E2 -28779.29} C_VEL
LIN {X 0,Y 100.38,Z 613.519,A -85,B 0,C 180,E1 -28783.737,E2 -28783.737} C_VEL
LIN {X 0,Y 109.994,Z 607.184,A -85,B 0,C 180,E1 -28786.996,E2 -28786.996} C_VEL
LIN {X 0,Y 120.067,Z 599.09,A -85,B 0,C 180,E1 -28789.722,E2 -28789.722} C_VEL
LIN {X 0,Y 129.546,Z 589.615,A -85,B 0,C 180,E1 -28791.908,E2 -28791.908} C_VEL
LIN {X 0,Y 137.925,Z 579.422,A -85,B 0,C 180,E1 -28793.511,E2 -28793.511} C_VEL
LIN {X 0,Y 144.479,Z 569.62,A -85,B 0,C 180,E1 -28794.67,E2 -28794.67} C_VEL
LIN {X 0,Y 150.626,Z 558.212,A -85,B 0,C 180,E1 -28795.63,E2 -28795.63} C_VEL
LIN {X 0,Y 155.501,Z 546.635,A -85,B 0,C 180,E1 -28796.33,E2 -28796.33} C_VEL
LIN {X 0,Y 157.928,Z 539.439,A -85,B 0,C 180,E1 -28796.653,E2 -28796.653} C_VEL
LIN {X 0,Y 158.394,Z 537.638,A -85,B 0,C 180,E1 -28796.821,E2 -28796.821} C_VEL
LIN {X 0,Y 158.075,Z 535.387,A -85,B 0,C 180,E1 -28799.204,E2 -28799.204} C_VEL
LIN {X 0,Y 157.857,Z 533.693,A -85,B 0,C 180,E1 -28801.595,E2 -28801.595} C_VEL
LIN {X 0,Y 157.602,Z 532.56,A -85,B 0,C 180,E1 -28805.117,E2 -28805.117} C_VEL
LIN {X 0,Y 157.555,Z 533.359,A -85,B 0,C 180,E1 -28808.982,E2 -28808.982} C_VEL
LIN {X 0,Y 157.92,Z 534.548,A -85,B 0,C 180,E1 -28812.14,E2 -28812.14} C_VEL
LIN {X 0,Y 158.453,Z 537.643,A -85,B 0,C 180,E1 -28815.89,E2 -28815.89} C_VEL
LIN {X 0,Y 158.416,Z 538.206,A -85,B 0,C 180,E1 -28816.157,E2 -28816.157} C_VEL
LIN {X 0,Y 154.1,Z 550.919,A -85,B 0,C 180,E1 -28816.723,E2 -28816.723} C_VEL
LIN {X 0,Y 148.278,Z 563.457,A -85,B 0,C 180,E1 -28817.517,E2 -28817.517} C_VEL
LIN {X 0,Y 141.692,Z 574.562,A -85,B 0,C 180,E1 -28818.454,E2 -28818.454} C_VEL
LIN {X 0,Y 134.384,Z 584.609,A -85,B 0,C 180,E1 -28819.724,E2 -28819.724} C_VEL
LIN {X 0,Y 126.385,Z 593.673,A -85,B 0,C 180,E1 -28821.346,E2 -28821.346} C_VEL
LIN {X 0,Y 116.932,Z 602.525,A -85,B 0,C 180,E1 -28823.574,E2 -28823.574} C_VEL
LIN {X 0,Y 107.616,Z 609.68,A -85,B 0,C 180,E1 -28826.113,E2 -28826.113} C_VEL
LIN {X 0,Y 97.195,Z 616.215,A -85,B 0,C 180,E1 -28829.812,E2 -28829.812} C_VEL
LIN {X 0,Y 89.785,Z 620.092,A -85,B 0,C 180,E1 -28833.226,E2 -28833.226} C_VEL
LIN {X 0,Y 80.776,Z 623.856,A -85,B 0,C 180,E1 -28838.462,E2 -28838.462} C_VEL
LIN {X 0,Y 71.179,Z 626.769,A -85,B 0,C 180,E1 -28846.281,E2 -28846.281} C_VEL
LIN {X 0,Y 66.972,Z 627.645,A -85,B 0,C 180,E1 -28850.98,E2 -28850.98} C_VEL
LIN {X 0,Y 63.302,Z 628.1,A -85,B 0,C 180,E1 -28856.284,E2 -28856.284} C_VEL
LIN {X 0,Y 58.033,Z 627.87,A -85,B 0,C 180,E1 -28868.699,E2 -28868.699} C_VEL
LIN {X 0,Y 56.452,Z 627.192,A -85,B 0,C 180,E1 -28875.584,E2 -28875.584} C_VEL
LIN {X 0,Y 55.607,Z 626.104,A -85,B 0,C 180,E1 -28882.741,E2 -28882.741} C_VEL
LIN {X 0,Y 55.465,Z 624.581,A -85,B 0,C 180,E1 -28890.002,E2 -28890.002} C_VEL
LIN {X 0,Y 55.823,Z 621.466,A -85,B 0,C 180,E1 -28900.887,E2 -28900.887} C_VEL
LIN {X 0,Y 57.769,Z 617.263,A -85,B 0,C 180,E1 -28911.407,E2 -28911.407} C_VEL
LIN {X 0,Y 62.032,Z 610.832,A -85,B 0,C 180,E1 -28922.559,E2 -28922.559} C_VEL
LIN {X 0,Y 67.316,Z 603.803,A -85,B 0,C 180,E1 -28930.733,E2 -28930.733} C_VEL
LIN {X 0,Y 72.253,Z 597.023,A -85,B 0,C 180,E1 -28936.302,E2 -28936.302} C_VEL
LIN {X 0,Y 77.124,Z 589.731,A -85,B 0,C 180,E1 -28940.767,E2 -28940.767} C_VEL
LIN {X 0,Y 83.36,Z 579.405,A -85,B 0,C 180,E1 -28945.287,E2 -28945.287} C_VEL
LIN {X 0,Y 87.314,Z 571.93,A -85,B 0,C 180,E1 -28947.689,E2 -28947.689} C_VEL
LIN {X 0,Y 92.235,Z 561.514,A -85,B 0,C 180,E1 -28950.082,E2 -28950.082} C_VEL
LIN {X 0,Y 96.461,Z 550.066,A -85,B 0,C 180,E1 -28952.057,E2 -28952.057} C_VEL
LIN {X 0,Y 100.239,Z 536.381,A -85,B 0,C 180,E1 -28953.653,E2 -28953.653} C_VEL
LIN {X 0,Y 102.623,Z 523.698,A -85,B 0,C 180,E1 -28954.549,E2 -28954.549} C_VEL
LIN {X 0,Y 105.794,Z 492.964,A -85,B 0,C 180,E1 -28955.865,E2 -28955.865} C_VEL
LIN {X 0,Y 103.74,Z 487.665,A -85,B 0,C 180,E1 -28958.645,E2 -28958.645} C_VEL
LIN {X 0,Y 100.938,Z 481.437,A -85,B 0,C 180,E1 -28962.918,E2 -28962.918} C_VEL
LIN {X 0,Y 98.047,Z 475.79,A -85,B 0,C 180,E1 -28968.438,E2 -28968.438} C_VEL
LIN {X 0,Y 96.181,Z 472.054,A -85,B 0,C 180,E1 -28973.414,E2 -28973.414} C_VEL
LIN {X 0,Y 94.714,Z 468.967,A -85,B 0,C 180,E1 -28979.829,E2 -28979.829} C_VEL
LIN {X 0,Y 94.572,Z 468.143,A -85,B 0,C 180,E1 -28981.255,E2 -28981.255} C_VEL
LIN {X 0,Y 94.441,Z 468.375,A -85,B 0,C 180,E1 -28991.264,E2 -28991.264} C_VEL
LIN {X 0,Y 95.342,Z 471.309,A -85,B 0,C 180,E1 -28997.148,E2 -28997.148} C_VEL
LIN {X 0,Y 96.57,Z 473.125,A -85,B 0,C 180,E1 -29001.126,E2 -29001.126} C_VEL
LIN {X 0,Y 98.632,Z 477.149,A -85,B 0,C 180,E1 -29006.136,E2 -29006.136} C_VEL
LIN {X 0,Y 101.386,Z 482.468,A -85,B 0,C 180,E1 -29011.092,E2 -29011.092} C_VEL
LIN {X 0,Y 104.543,Z 489.527,A -85,B 0,C 180,E1 -29015.708,E2 -29015.708} C_VEL
LIN {X 0,Y 104.807,Z 490.244,A -85,B 0,C 180,E1 -29016.073,E2 -29016.073} C_VEL
LIN {X 0,Y 105.048,Z 492.751,A -85,B 0,C 180,E1 -29016.656,E2 -29016.656} C_VEL
LIN {X 0,Y 104.568,Z 496.222,A -85,B 0,C 180,E1 -29016.671,E2 -29016.671} C_VEL
LIN {X 0,Y 103.518,Z 499.961,A -85,B 0,C 180,E1 -29016.165,E2 -29016.165} C_VEL
LIN {X 0,Y 101.319,Z 506.678,A -85,B 0,C 180,E1 -29014.872,E2 -29014.872} C_VEL
LIN {X 0,Y 100.49,Z 510.94,A -85,B 0,C 180,E1 -29014.626,E2 -29014.626} C_VEL
LIN {X 0,Y 98.355,Z 527.065,A -85,B 0,C 180,E1 -29015.332,E2 -29015.332} C_VEL
LIN {X 0,Y 95.58,Z 539.473,A -85,B 0,C 180,E1 -29016.367,E2 -29016.367} C_VEL
LIN {X 0,Y 92.072,Z 550.654,A -85,B 0,C 180,E1 -29017.749,E2 -29017.749} C_VEL
LIN {X 0,Y 87.117,Z 562.893,A -85,B 0,C 180,E1 -29019.969,E2 -29019.969} C_VEL
LIN {X 0,Y 81.394,Z 574.07,A -85,B 0,C 180,E1 -29022.782,E2 -29022.782} C_VEL
LIN {X 0,Y 76.584,Z 582.038,A -85,B 0,C 180,E1 -29025.593,E2 -29025.593} C_VEL
LIN {X 0,Y 70.695,Z 590.665,A -85,B 0,C 180,E1 -29029.745,E2 -29029.745} C_VEL
LIN {X 0,Y 64.773,Z 598.593,A -85,B 0,C 180,E1 -29035.274,E2 -29035.274} C_VEL
LIN {X 0,Y 58.422,Z 606.352,A -85,B 0,C 180,E1 -29043.183,E2 -29043.183} C_VEL
LIN {X 0,Y 54.175,Z 611.648,A -85,B 0,C 180,E1 -29051.074,E2 -29051.074} C_VEL
LIN {X 0,Y 50.466,Z 616.782,A -85,B 0,C 180,E1 -29061.993,E2 -29061.993} C_VEL
LIN {X 0,Y 48.261,Z 620.788,A -85,B 0,C 180,E1 -29074.173,E2 -29074.173} C_VEL
LIN {X 0,Y 47.839,Z 623.755,A -85,B 0,C 180,E1 -29087.084,E2 -29087.084} C_VEL
LIN {X 0,Y 48.757,Z 625.155,A -85,B 0,C 180,E1 -29095.619,E2 -29095.619} C_VEL
LIN {X 0,Y 50.549,Z 626.152,A -85,B 0,C 180,E1 -29103.786,E2 -29103.786} C_VEL
LIN {X 0,Y 53.172,Z 626.747,A -85,B 0,C 180,E1 -29111.363,E2 -29111.363} C_VEL
LIN {X 0,Y 56.607,Z 626.885,A -85,B 0,C 180,E1 -29118.149,E2 -29118.149} C_VEL
LIN {X 0,Y 61.626,Z 626.509,A -85,B 0,C 180,E1 -29125.236,E2 -29125.236} C_VEL
LIN {X 0,Y 70.505,Z 624.815,A -85,B 0,C 180,E1 -29133.778,E2 -29133.778} C_VEL
LIN {X 0,Y 78.181,Z 622.535,A -85,B 0,C 180,E1 -29138.926,E2 -29138.926} C_VEL
LIN {X 0,Y 87.81,Z 618.722,A -85,B 0,C 180,E1 -29143.821,E2 -29143.821} C_VEL
LIN {X 0,Y 97.514,Z 613.791,A -85,B 0,C 180,E1 -29147.514,E2 -29147.514} C_VEL
LIN {X 0,Y 106.926,Z 607.889,A -85,B 0,C 180,E1 -29150.358,E2 -29150.358} C_VEL
LIN {X 0,Y 116.257,Z 600.802,A -85,B 0,C 180,E1 -29152.615,E2 -29152.615} C_VEL
LIN {X 0,Y 125.318,Z 592.453,A -85,B 0,C 180,E1 -29154.508,E2 -29154.508} C_VEL
LIN {X 0,Y 133.853,Z 582.887,A -85,B 0,C 180,E1 -29156.002,E2 -29156.002} C_VEL
LIN {X 0,Y 141.087,Z 572.945,A -85,B 0,C 180,E1 -29157.145,E2 -29157.145} C_VEL
LIN {X 0,Y 147.667,Z 561.798,A -85,B 0,C 180,E1 -29158.064,E2 -29158.064} C_VEL
LIN {X 0,Y 152.449,Z 551.656,A -85,B 0,C 180,E1 -29158.661,E2 -29158.661} C_VEL
LIN {X 0,Y 155.891,Z 542.458,A -85,B 0,C 180,E1 -29159.099,E2 -29159.099} C_VEL
LIN {X 0,Y 155.743,Z 540.172,A -85,B 0,C 180,E1 -29162.587,E2 -29162.587} C_VEL
LIN {X 0,Y 155.685,Z 539.401,A -85,B 0,C 180,E1 -29165.18,E2 -29165.18} C_VEL
LIN {X 0,Y 155.687,Z 540.614,A -85,B 0,C 180,E1 -29170.403,E2 -29170.403} C_VEL
LIN {X 0,Y 155.889,Z 542.765,A -85,B 0,C 180,E1 -29173.691,E2 -29173.691} C_VEL
LIN {X 0,Y 154.222,Z 547.579,A -85,B 0,C 180,E1 -29173.964,E2 -29173.964} C_VEL
LIN {X 0,Y 148.66,Z 560.356,A -85,B 0,C 180,E1 -29174.625,E2 -29174.625} C_VEL
LIN {X 0,Y 142.141,Z 571.761,A -85,B 0,C 180,E1 -29175.394,E2 -29175.394} C_VEL
LIN {X 0,Y 135.494,Z 581.246,A -85,B 0,C 180,E1 -29176.352,E2 -29176.352} C_VEL
LIN {X 0,Y 127.248,Z 590.942,A -85,B 0,C 180,E1 -29177.693,E2 -29177.693} C_VEL
LIN {X 0,Y 119.134,Z 598.896,A -85,B 0,C 180,E1 -29179.293,E2 -29179.293} C_VEL
LIN {X 0,Y 109.471,Z 606.74,A -85,B 0,C 180,E1 -29181.43,E2 -29181.43} C_VEL
LIN {X 0,Y 100.012,Z 613.022,A -85,B 0,C 180,E1 -29184.008,E2 -29184.008} C_VEL
LIN {X 0,Y 90.889,Z 618.033,A -85,B 0,C 180,E1 -29187.227,E2 -29187.227} C_VEL
LIN {X 0,Y 82.15,Z 621.937,A -85,B 0,C 180,E1 -29191.189,E2 -29191.189} C_VEL
LIN {X 0,Y 71.199,Z 625.571,A -85,B 0,C 180,E1 -29197.849,E2 -29197.849} C_VEL
LIN {X 0,Y 66.229,Z 626.794,A -85,B 0,C 180,E1 -29202.031,E2 -29202.031} C_VEL
LIN {X 0,Y 61.62,Z 627.609,A -85,B 0,C 180,E1 -29206.821,E2 -29206.821} C_VEL
LIN {X 0,Y 54.138,Z 628.054,A -85,B 0,C 180,E1 -29218.72,E2 -29218.72} C_VEL
LIN {X 0,Y 49.589,Z 626.999,A -85,B 0,C 180,E1 -29233.536,E2 -29233.536} C_VEL
LIN {X 0,Y 48.579,Z 625.848,A -85,B 0,C 180,E1 -29241.684,E2 -29241.684} C_VEL
LIN {X 0,Y 48.365,Z 624.289,A -85,B 0,C 180,E1 -29250.002,E2 -29250.002} C_VEL
LIN {X 0,Y 48.856,Z 621.099,A -85,B 0,C 180,E1 -29262.463,E2 -29262.463} C_VEL
LIN {X 0,Y 51.179,Z 616.815,A -85,B 0,C 180,E1 -29274.33,E2 -29274.33} C_VEL
LIN {X 0,Y 56.154,Z 610.298,A -85,B 0,C 180,E1 -29286.478,E2 -29286.478} C_VEL
LIN {X 0,Y 62.054,Z 603.122,A -85,B 0,C 180,E1 -29295.061,E2 -29295.061} C_VEL
LIN {X 0,Y 67.132,Z 596.697,A -85,B 0,C 180,E1 -29300.419,E2 -29300.419} C_VEL
LIN {X 0,Y 72.815,Z 588.86,A -85,B 0,C 180,E1 -29305.126,E2 -29305.126} C_VEL
LIN {X 0,Y 79.497,Z 578.293,A -85,B 0,C 180,E1 -29309.538,E2 -29309.538} C_VEL
LIN {X 0,Y 83.743,Z 570.71,A -85,B 0,C 180,E1 -29311.787,E2 -29311.787} C_VEL
LIN {X 0,Y 88.843,Z 559.912,A -85,B 0,C 180,E1 -29314.136,E2 -29314.136} C_VEL
LIN {X 0,Y 93.2,Z 548.305,A -85,B 0,C 180,E1 -29315.936,E2 -29315.936} C_VEL
LIN {X 0,Y 96.926,Z 535.136,A -85,B 0,C 180,E1 -29317.287,E2 -29317.287} C_VEL
LIN {X 0,Y 99.329,Z 521.905,A -85,B 0,C 180,E1 -29318.114,E2 -29318.114} C_VEL
LIN {X 0,Y 102.094,Z 495.669,A -85,B 0,C 180,E1 -29319.215,E2 -29319.215} C_VEL
LIN {X 0,Y 99.294,Z 488.604,A -85,B 0,C 180,E1 -29323.823,E2 -29323.823} C_VEL
LIN {X 0,Y 97.51,Z 484.689,A -85,B 0,C 180,E1 -29327.338,E2 -29327.338} C_VEL
LIN {X 0,Y 96.036,Z 481.567,A -85,B 0,C 180,E1 -29330.901,E2 -29330.901} C_VEL
LIN {X 0,Y 94.855,Z 478.732,A -85,B 0,C 180,E1 -29334.711,E2 -29334.711} C_VEL
LIN {X 0,Y 93.645,Z 475.548,A -85,B 0,C 180,E1 -29341.267,E2 -29341.267} C_VEL
LIN {X 0,Y 93.528,Z 475.157,A -85,B 0,C 180,E1 -29342.539,E2 -29342.539} C_VEL
LIN {X 0,Y 93.458,Z 475.366,A -85,B 0,C 180,E1 -29350.288,E2 -29350.288} C_VEL
LIN {X 0,Y 95.181,Z 479.75,A -85,B 0,C 180,E1 -29359.795,E2 -29359.795} C_VEL
LIN {X 0,Y 96.913,Z 483.546,A -85,B 0,C 180,E1 -29364.602,E2 -29364.602} C_VEL
LIN {X 0,Y 99.237,Z 488.562,A -85,B 0,C 180,E1 -29369.348,E2 -29369.348} C_VEL
LIN {X 0,Y 101.819,Z 494.913,A -85,B 0,C 180,E1 -29373.625,E2 -29373.625} C_VEL
LIN {X 0,Y 102.025,Z 495.603,A -85,B 0,C 180,E1 -29373.958,E2 -29373.958} C_VEL
LIN {X 0,Y 100.49,Z 510.94,A -85,B 0,C 180,E1 -29374.626,E2 -29374.626} C_VEL
LIN {X 0,Y 99.759,Z 514.848,A -85,B 0,C 180,E1 -29374.424,E2 -29374.424} C_VEL
LIN {X 0,Y 95.467,Z 526.955,A -85,B 0,C 180,E1 -29371.922,E2 -29371.922} C_VEL
LIN {X 0,Y 94.423,Z 530.795,A -85,B 0,C 180,E1 -29371.825,E2 -29371.825} C_VEL
LIN {X 0,Y 90.928,Z 543.958,A -85,B 0,C 180,E1 -29372.928,E2 -29372.928} C_VEL
LIN {X 0,Y 86.326,Z 556.57,A -85,B 0,C 180,E1 -29374.715,E2 -29374.715} C_VEL
LIN {X 0,Y 80.498,Z 568.81,A -85,B 0,C 180,E1 -29377.186,E2 -29377.186} C_VEL
LIN {X 0,Y 73.76,Z 579.939,A -85,B 0,C 180,E1 -29380.336,E2 -29380.336} C_VEL
LIN {X 0,Y 68.191,Z 588.017,A -85,B 0,C 180,E1 -29383.825,E2 -29383.825} C_VEL
LIN {X 0,Y 61.543,Z 596.413,A -85,B 0,C 180,E1 -29388.955,E2 -29388.955} C_VEL
LIN {X 0,Y 54.332,Z 604.624,A -85,B 0,C 180,E1 -29396.649,E2 -29396.649} C_VEL
LIN {X 0,Y 49.255,Z 610.209,A -85,B 0,C 180,E1 -29404.654,E2 -29404.654} C_VEL
LIN {X 0,Y 44.549,Z 615.669,A -85,B 0,C 180,E1 -29416.31,E2 -29416.31} C_VEL
LIN {X 0,Y 41.619,Z 619.953,A -85,B 0,C 180,E1 -29429.998,E2 -29429.998} C_VEL
LIN {X 0,Y 40.723,Z 622.241,A -85,B 0,C 180,E1 -29439.935,E2 -29439.935} C_VEL
LIN {X 0,Y 40.9,Z 624.035,A -85,B 0,C 180,E1 -29450.098,E2 -29450.098} C_VEL
LIN {X 0,Y 43.947,Z 626.149,A -85,B 0,C 180,E1 -29466.91,E2 -29466.91} C_VEL
LIN {X 0,Y 47.855,Z 626.885,A -85,B 0,C 180,E1 -29477.244,E2 -29477.244} C_VEL
LIN {X 0,Y 51.953,Z 626.97,A -85,B 0,C 180,E1 -29484.253,E2 -29484.253} C_VEL
LIN {X 0,Y 56.798,Z 626.642,A -85,B 0,C 180,E1 -29490.334,E2 -29490.334} C_VEL
LIN {X 0,Y 61.924,Z 625.93,A -85,B 0,C 180,E1 -29495.218,E2 -29495.218} C_VEL
LIN {X 0,Y 67.556,Z 624.741,A -85,B 0,C 180,E1 -29499.429,E2 -29499.429} C_VEL
LIN {X 0,Y 74.713,Z 622.752,A -85,B 0,C 180,E1 -29503.609,E2 -29503.609} C_VEL
LIN {X 0,Y 86.04,Z 618.476,A -85,B 0,C 180,E1 -29508.565,E2 -29508.565} C_VEL
LIN {X 0,Y 96.709,Z 613.158,A -85,B 0,C 180,E1 -29511.97,E2 -29511.97} C_VEL
LIN {X 0,Y 107.638,Z 606.299,A -85,B 0,C 180,E1 -29514.672,E2 -29514.672} C_VEL
LIN {X 0,Y 117.271,Z 598.792,A -85,B 0,C 180,E1 -29516.565,E2 -29516.565} C_VEL
LIN {X 0,Y 126.567,Z 589.923,A -85,B 0,C 180,E1 -29518.13,E2 -29518.13} C_VEL
LIN {X 0,Y 135.115,Z 579.973,A -85,B 0,C 180,E1 -29519.354,E2 -29519.354} C_VEL
LIN {X 0,Y 142.314,Z 569.635,A -85,B 0,C 180,E1 -29520.301,E2 -29520.301} C_VEL
LIN {X 0,Y 149.152,Z 557.189,A -85,B 0,C 180,E1 -29521.088,E2 -29521.088} C_VEL
LIN {X 0,Y 153.025,Z 548.316,A -85,B 0,C 180,E1 -29521.475,E2 -29521.475} C_VEL
LIN {X 0,Y 153.279,Z 547.56,A -85,B 0,C 180,E1 -29521.655,E2 -29521.655} C_VEL
LIN {X 0,Y 153.354,Z 546.109,A -85,B 0,C 180,E1 -29525.259,E2 -29525.259} C_VEL
LIN {X 0,Y 153.222,Z 546.581,A -85,B 0,C 180,E1 -29527.909,E2 -29527.909} C_VEL
LIN {X 0,Y 153.24,Z 547.779,A -85,B 0,C 180,E1 -29530.97,E2 -29530.97} C_VEL
LIN {X 0,Y 152.885,Z 548.941,A -85,B 0,C 180,E1 -29531.384,E2 -29531.384} C_VEL
LIN {X 0,Y 147.492,Z 560.872,A -85,B 0,C 180,E1 -29531.928,E2 -29531.928} C_VEL
LIN {X 0,Y 140.43,Z 572.815,A -85,B 0,C 180,E1 -29532.613,E2 -29532.613} C_VEL
LIN {X 0,Y 132.84,Z 583.159,A -85,B 0,C 180,E1 -29533.563,E2 -29533.563} C_VEL
LIN {X 0,Y 125.287,Z 591.635,A -85,B 0,C 180,E1 -29534.623,E2 -29534.623} C_VEL
LIN {X 0,Y 116.992,Z 599.459,A -85,B 0,C 180,E1 -29536.029,E2 -29536.029} C_VEL
LIN {X 0,Y 107.091,Z 607.148,A -85,B 0,C 180,E1 -29537.909,E2 -29537.909} C_VEL
LIN {X 0,Y 97.341,Z 613.328,A -85,B 0,C 180,E1 -29540.189,E2 -29540.189} C_VEL
LIN {X 0,Y 87.866,Z 618.252,A -85,B 0,C 180,E1 -29543.103,E2 -29543.103} C_VEL
LIN {X 0,Y 78.7,Z 622.076,A -85,B 0,C 180,E1 -29546.75,E2 -29546.75} C_VEL
LIN {X 0,Y 72.807,Z 624.055,A -85,B 0,C 180,E1 -29549.69,E2 -29549.69} C_VEL
LIN {X 0,Y 67.072,Z 625.634,A -85,B 0,C 180,E1 -29553.048,E2 -29553.048} C_VEL
LIN {X 0,Y 61.691,Z 626.811,A -85,B 0,C 180,E1 -29557.116,E2 -29557.116} C_VEL
LIN {X 0,Y 52.053,Z 627.934,A -85,B 0,C 180,E1 -29567.543,E2 -29567.543} C_VEL
LIN {X 0,Y 45.073,Z 627.563,A -85,B 0,C 180,E1 -29582.113,E2 -29582.113} C_VEL
LIN {X 0,Y 42.821,Z 626.779,A -85,B 0,C 180,E1 -29590.84,E2 -29590.84} C_VEL
LIN {X 0,Y 41.583,Z 625.587,A -85,B 0,C 180,E1 -29600.272,E2 -29600.272} C_VEL
LIN {X 0,Y 41.282,Z 623.993,A -85,B 0,C 180,E1 -29610.002,E2 -29610.002} C_VEL
LIN {X 0,Y 41.951,Z 620.726,A -85,B 0,C 180,E1 -29624.556,E2 -29624.556} C_VEL
LIN {X 0,Y 44.771,Z 616.357,A -85,B 0,C 180,E1 -29638.097,E2 -29638.097} C_VEL
LIN {X 0,Y 49.61,Z 610.77,A -85,B 0,C 180,E1 -29649.607,E2 -29649.607} C_VEL
LIN {X 0,Y 56.047,Z 603.777,A -85,B 0,C 180,E1 -29658.798,E2 -29658.798} C_VEL
LIN {X 0,Y 62.075,Z 596.79,A -85,B 0,C 180,E1 -29664.837,E2 -29664.837} C_VEL
LIN {X 0,Y 68.981,Z 587.905,A -85,B 0,C 180,E1 -29669.998,E2 -29669.998} C_VEL
LIN {X 0,Y 76.094,Z 577.131,A -85,B 0,C 180,E1 -29674.225,E2 -29674.225} C_VEL
LIN {X 0,Y 82.119,Z 566.45,A -85,B 0,C 180,E1 -29676.93,E2 -29676.93} C_VEL
LIN {X 0,Y 87.529,Z 554.511,A -85,B 0,C 180,E1 -29678.972,E2 -29678.972} C_VEL
LIN {X 0,Y 91.511,Z 543.063,A -85,B 0,C 180,E1 -29680.36,E2 -29680.36} C_VEL
LIN {X 0,Y 94.805,Z 529.994,A -85,B 0,C 180,E1 -29681.403,E2 -29681.403} C_VEL
LIN {X 0,Y 96.794,Z 516.718,A -85,B 0,C 180,E1 -29682.062,E2 -29682.062} C_VEL
LIN {X 0,Y 98.687,Z 498.751,A -85,B 0,C 180,E1 -29682.788,E2 -29682.788} C_VEL
LIN {X 0,Y 96.595,Z 492.976,A -85,B 0,C 180,E1 -29687.04,E2 -29687.04} C_VEL
LIN {X 0,Y 94.607,Z 488.174,A -85,B 0,C 180,E1 -29692.206,E2 -29692.206} C_VEL
LIN {X 0,Y 93.478,Z 485.244,A -85,B 0,C 180,E1 -29696.458,E2 -29696.458} C_VEL
LIN {X 0,Y 92.604,Z 482.202,A -85,B 0,C 180,E1 -29702.976,E2 -29702.976} C_VEL
LIN {X 0,Y 92.537,Z 482.522,A -85,B 0,C 180,E1 -29709.976,E2 -29709.976} C_VEL
LIN {X 0,Y 93.891,Z 486.514,A -85,B 0,C 180,E1 -29718.617,E2 -29718.617} C_VEL
LIN {X 0,Y 95.277,Z 489.954,A -85,B 0,C 180,E1 -29723.04,E2 -29723.04} C_VEL
LIN {X 0,Y 97.367,Z 495.105,A -85,B 0,C 180,E1 -29727.904,E2 -29727.904} C_VEL
LIN {X 0,Y 98.638,Z 498.616,A -85,B 0,C 180,E1 -29730.382,E2 -29730.382} C_VEL
LIN {X 0,Y 98.093,Z 504.461,A -85,B 0,C 180,E1 -29730.711,E2 -29730.711} C_VEL
LIN {X 0,Y 95.676,Z 524.105,A -85,B 0,C 180,E1 -29731.403,E2 -29731.403} C_VEL
LIN {X 0,Y 94.423,Z 530.795,A -85,B 0,C 180,E1 -29731.825,E2 -29731.825} C_VEL
LIN {X 0,Y 93.443,Z 534.601,A -85,B 0,C 180,E1 -29731.944,E2 -29731.944} C_VEL
LIN {X 0,Y 90.623,Z 541.958,A -85,B 0,C 180,E1 -29731.487,E2 -29731.487} C_VEL
LIN {X 0,Y 84.481,Z 554.339,A -85,B 0,C 180,E1 -29730.437,E2 -29730.437} C_VEL
LIN {X 0,Y 81.914,Z 559.629,A -85,B 0,C 180,E1 -29730.862,E2 -29730.862} C_VEL
LIN {X 0,Y 75.606,Z 571.515,A -85,B 0,C 180,E1 -29733.217,E2 -29733.217} C_VEL
LIN {X 0,Y 70.132,Z 579.972,A -85,B 0,C 180,E1 -29735.489,E2 -29735.489} C_VEL
LIN {X 0,Y 63.469,Z 588.96,A -85,B 0,C 180,E1 -29739.183,E2 -29739.183} C_VEL
LIN {X 0,Y 56.372,Z 597.215,A -85,B 0,C 180,E1 -29744.203,E2 -29744.203} C_VEL
LIN {X 0,Y 48.525,Z 605.309,A -85,B 0,C 180,E1 -29752.007,E2 -29752.007} C_VEL
LIN {X 0,Y 42.925,Z 610.786,A -85,B 0,C 180,E1 -29760.579,E2 -29760.579} C_VEL
LIN {X 0,Y 37.649,Z 616.152,A -85,B 0,C 180,E1 -29773.737,E2 -29773.737} C_VEL
LIN {X 0,Y 34.384,Z 620.354,A -85,B 0,C 180,E1 -29789.997,E2 -29789.997} C_VEL
LIN {X 0,Y 33.566,Z 622.577,A -85,B 0,C 180,E1 -29802.083,E2 -29802.083} C_VEL
LIN {X 0,Y 34.116,Z 624.314,A -85,B 0,C 180,E1 -29814.327,E2 -29814.327} C_VEL
LIN {X 0,Y 37.736,Z 626.205,A -85,B 0,C 180,E1 -29831.846,E2 -29831.846} C_VEL
LIN {X 0,Y 43.18,Z 627.009,A -85,B 0,C 180,E1 -29844.463,E2 -29844.463} C_VEL
LIN {X 0,Y 52.55,Z 626.77,A -85,B 0,C 180,E1 -29856.346,E2 -29856.346} C_VEL
LIN {X 0,Y 59.201,Z 625.912,A -85,B 0,C 180,E1 -29861.743,E2 -29861.743} C_VEL
LIN {X 0,Y 65.319,Z 624.667,A -85,B 0,C 180,E1 -29865.535,E2 -29865.535} C_VEL
LIN {X 0,Y 74.599,Z 622.097,A -85,B 0,C 180,E1 -29869.885,E2 -29869.885} C_VEL
LIN {X 0,Y 84.884,Z 618.231,A -85,B 0,C 180,E1 -29873.464,E2 -29873.464} C_VEL
LIN {X 0,Y 95.055,Z 613.306,A -85,B 0,C 180,E1 -29876.135,E2 -29876.135} C_VEL
LIN {X 0,Y 105.463,Z 607.004,A -85,B 0,C 180,E1 -29878.287,E2 -29878.287} C_VEL
LIN {X 0,Y 116,Z 599.092,A -85,B 0,C 180,E1 -29880,E2 -29880} C_VEL
LIN {X 0,Y 124.771,Z 590.991,A -85,B 0,C 180,E1 -29881.231,E2 -29881.231} C_VEL
LIN {X 0,Y 133.634,Z 581.014,A -85,B 0,C 180,E1 -29882.283,E2 -29882.283} C_VEL
LIN {X 0,Y 141.648,Z 569.822,A -85,B 0,C 180,E1 -29883.15,E2 -29883.15} C_VEL
LIN {X 0,Y 148.568,Z 557.41,A -85,B 0,C 180,E1 -29883.816,E2 -29883.816} C_VEL
LIN {X 0,Y 150.566,Z 553.103,A -85,B 0,C 180,E1 -29884.057,E2 -29884.057} C_VEL
LIN {X 0,Y 150.642,Z 552.714,A -85,B 0,C 180,E1 -29885.354,E2 -29885.354} C_VEL
LIN {X 0,Y 150.459,Z 553.392,A -85,B 0,C 180,E1 -29888.477,E2 -29888.477} C_VEL
LIN {X 0,Y 150.261,Z 553.958,A -85,B 0,C 180,E1 -29888.899,E2 -29888.899} C_VEL
LIN {X 0,Y 144.396,Z 565.451,A -85,B 0,C 180,E1 -29889.355,E2 -29889.355} C_VEL
LIN {X 0,Y 137.344,Z 576.303,A -85,B 0,C 180,E1 -29889.934,E2 -29889.934} C_VEL
LIN {X 0,Y 128.79,Z 586.922,A -85,B 0,C 180,E1 -29890.821,E2 -29890.821} C_VEL
LIN {X 0,Y 120.303,Z 595.553,A -85,B 0,C 180,E1 -29891.907,E2 -29891.907} C_VEL
LIN {X 0,Y 110.172,Z 603.976,A -85,B 0,C 180,E1 -29893.4,E2 -29893.4} C_VEL
LIN {X 0,Y 98.443,Z 611.76,A -85,B 0,C 180,E1 -29895.475,E2 -29895.475} C_VEL
LIN {X 0,Y 88.556,Z 617.001,A -85,B 0,C 180,E1 -29897.767,E2 -29897.767} C_VEL
LIN {X 0,Y 77.825,Z 621.514,A -85,B 0,C 180,E1 -29901.176,E2 -29901.176} C_VEL
LIN {X 0,Y 69.558,Z 624.156,A -85,B 0,C 180,E1 -29904.592,E2 -29904.592} C_VEL
LIN {X 0,Y 63.478,Z 625.696,A -85,B 0,C 180,E1 -29907.665,E2 -29907.665} C_VEL
LIN {X 0,Y 52.154,Z 627.516,A -85,B 0,C 180,E1 -29916.053,E2 -29916.053} C_VEL
LIN {X 0,Y 42.6,Z 627.816,A -85,B 0,C 180,E1 -29928.712,E2 -29928.712} C_VEL
LIN {X 0,Y 38.937,Z 627.394,A -85,B 0,C 180,E1 -29937.219,E2 -29937.219} C_VEL
LIN {X 0,Y 34.608,Z 625.324,A -85,B 0,C 180,E1 -29958.286,E2 -29958.286} C_VEL
LIN {X 0,Y 34.175,Z 623.691,A -85,B 0,C 180,E1 -29970.003,E2 -29970.003} C_VEL
LIN {X 0,Y 35.103,Z 620.345,A -85,B 0,C 180,E1 -29987.479,E2 -29987.479} C_VEL
LIN {X 0,Y 38.629,Z 615.893,A -85,B 0,C 180,E1 -30003.082,E2 -30003.082} C_VEL
LIN {X 0,Y 44.348,Z 610.214,A -85,B 0,C 180,E1 -30015.492,E2 -30015.492} C_VEL
LIN {X 0,Y 51.61,Z 603.075,A -85,B 0,C 180,E1 -30024.792,E2 -30024.792} C_VEL
LIN {X 0,Y 57.034,Z 597.35,A -85,B 0,C 180,E1 -30029.608,E2 -30029.608} C_VEL
LIN {X 0,Y 61.476,Z 592.18,A -85,B 0,C 180,E1 -30032.94,E2 -30032.94} C_VEL
LIN {X 0,Y 69.465,Z 581.753,A -85,B 0,C 180,E1 -30037.4,E2 -30037.4} C_VEL
LIN {X 0,Y 75.616,Z 572.109,A -85,B 0,C 180,E1 -30040.23,E2 -30040.23} C_VEL
LIN {X 0,Y 81.218,Z 561.798,A -85,B 0,C 180,E1 -30042.15,E2 -30042.15} C_VEL
LIN {X 0,Y 86.426,Z 549.451,A -85,B 0,C 180,E1 -30043.856,E2 -30043.856} C_VEL
LIN {X 0,Y 90.525,Z 536.281,A -85,B 0,C 180,E1 -30045.034,E2 -30045.034} C_VEL
LIN {X 0,Y 93.281,Z 522.922,A -85,B 0,C 180,E1 -30045.768,E2 -30045.768} C_VEL
LIN {X 0,Y 95.675,Z 502.07,A -85,B 0,C 180,E1 -30046.573,E2 -30046.573} C_VEL
LIN {X 0,Y 94.275,Z 497.725,A -85,B 0,C 180,E1 -30050.208,E2 -30050.208} C_VEL
LIN {X 0,Y 92.988,Z 494.196,A -85,B 0,C 180,E1 -30054.427,E2 -30054.427} C_VEL
LIN {X 0,Y 92.331,Z 492.012,A -85,B 0,C 180,E1 -30057.544,E2 -30057.544} C_VEL
LIN {X 0,Y 91.657,Z 489.249,A -85,B 0,C 180,E1 -30063.772,E2 -30063.772} C_VEL
LIN {X 0,Y 91.603,Z 489.438,A -85,B 0,C 180,E1 -30069.014,E2 -30069.014} C_VEL
LIN {X 0,Y 92.635,Z 493.282,A -85,B 0,C 180,E1 -30077.381,E2 -30077.381} C_VEL
LIN {X 0,Y 93.896,Z 496.823,A -85,B 0,C 180,E1 -30081.977,E2 -30081.977} C_VEL
LIN {X 0,Y 95.585,Z 501.771,A -85,B 0,C 180,E1 -30086.47,E2 -30086.47} C_VEL
LIN {X 0,Y 95.689,Z 502.325,A -85,B 0,C 180,E1 -30086.764,E2 -30086.764} C_VEL
LIN {X 0,Y 92.986,Z 523.94,A -85,B 0,C 180,E1 -30087.423,E2 -30087.423} C_VEL
LIN {X 0,Y 90.015,Z 537.51,A -85,B 0,C 180,E1 -30088.282,E2 -30088.282} C_VEL
LIN {X 0,Y 86.393,Z 548.781,A -85,B 0,C 180,E1 -30089.324,E2 -30089.324} C_VEL
LIN {X 0,Y 81.914,Z 559.629,A -85,B 0,C 180,E1 -30090.862,E2 -30090.862} C_VEL
LIN {X 0,Y 79.167,Z 564.814,A -85,B 0,C 180,E1 -30091.308,E2 -30091.308} C_VEL
LIN {X 0,Y 73.422,Z 572.88,A -85,B 0,C 180,E1 -30090.996,E2 -30090.996} C_VEL
LIN {X 0,Y 67.064,Z 580.482,A -85,B 0,C 180,E1 -30090.878,E2 -30090.878} C_VEL
LIN {X 0,Y 63.358,Z 584.941,A -85,B 0,C 180,E1 -30091.848,E2 -30091.848} C_VEL
LIN {X 0,Y 56.144,Z 593.339,A -85,B 0,C 180,E1 -30095.544,E2 -30095.544} C_VEL
LIN {X 0,Y 47.289,Z 602.223,A -85,B 0,C 180,E1 -30102.002,E2 -30102.002} C_VEL
LIN {X 0,Y 39.279,Z 609.332,A -85,B 0,C 180,E1 -30111.225,E2 -30111.225} C_VEL
LIN {X 0,Y 32.594,Z 615.006,A -85,B 0,C 180,E1 -30124.45,E2 -30124.45} C_VEL
LIN {X 0,Y 28.504,Z 619.045,A -85,B 0,C 180,E1 -30140.474,E2 -30140.474} C_VEL
LIN {X 0,Y 26.461,Z 622.897,A -85,B 0,C 180,E1 -30165.398,E2 -30165.398} C_VEL
LIN {X 0,Y 27.618,Z 624.594,A -85,B 0,C 180,E1 -30180.588,E2 -30180.588} C_VEL
LIN {X 0,Y 31.888,Z 626.258,A -85,B 0,C 180,E1 -30198.61,E2 -30198.61} C_VEL
LIN {X 0,Y 39.33,Z 627.134,A -85,B 0,C 180,E1 -30213.305,E2 -30213.305} C_VEL
LIN {X 0,Y 48.904,Z 626.904,A -85,B 0,C 180,E1 -30223.297,E2 -30223.297} C_VEL
LIN {X 0,Y 57.31,Z 625.879,A -85,B 0,C 180,E1 -30228.812,E2 -30228.812} C_VEL
LIN {X 0,Y 69.574,Z 623.16,A -85,B 0,C 180,E1 -30234.203,E2 -30234.203} C_VEL
LIN {X 0,Y 80.888,Z 619.414,A -85,B 0,C 180,E1 -30237.621,E2 -30237.621} C_VEL
LIN {X 0,Y 91.715,Z 614.617,A -85,B 0,C 180,E1 -30240,E2 -30240} C_VEL
LIN {X 0,Y 101.949,Z 608.859,A -85,B 0,C 180,E1 -30241.743,E2 -30241.743} C_VEL
LIN {X 0,Y 112.616,Z 601.389,A -85,B 0,C 180,E1 -30243.172,E2 -30243.172} C_VEL
LIN {X 0,Y 121.56,Z 593.731,A -85,B 0,C 180,E1 -30244.233,E2 -30244.233} C_VEL
LIN {X 0,Y 130.528,Z 584.42,A -85,B 0,C 180,E1 -30245.09,E2 -30245.09} C_VEL
LIN {X 0,Y 138.68,Z 573.944,A -85,B 0,C 180,E1 -30245.818,E2 -30245.818} C_VEL
LIN {X 0,Y 141.335,Z 570.007,A -85,B 0,C 180,E1 -30246.023,E2 -30246.023} C_VEL
LIN {X 0,Y 141.518,Z 569.732,A -85,B 0,C 180,E1 -30246.687,E2 -30246.687} C_VEL
LIN {X 0,Y 133.708,Z 580.631,A -85,B 0,C 180,E1 -30247.215,E2 -30247.215} C_VEL
LIN {X 0,Y 125.938,Z 589.489,A -85,B 0,C 180,E1 -30247.9,E2 -30247.9} C_VEL
LIN {X 0,Y 117.339,Z 597.637,A -85,B 0,C 180,E1 -30248.799,E2 -30248.799} C_VEL
LIN {X 0,Y 107.036,Z 605.651,A -85,B 0,C 180,E1 -30249.982,E2 -30249.982} C_VEL
LIN {X 0,Y 96.796,Z 612.111,A -85,B 0,C 180,E1 -30251.436,E2 -30251.436} C_VEL
LIN {X 0,Y 86.656,Z 617.26,A -85,B 0,C 180,E1 -30253.297,E2 -30253.297} C_VEL
LIN {X 0,Y 74.545,Z 621.984,A -85,B 0,C 180,E1 -30256.43,E2 -30256.43} C_VEL
LIN {X 0,Y 66.911,Z 624.256,A -85,B 0,C 180,E1 -30259.044,E2 -30259.044} C_VEL
LIN {X 0,Y 60.508,Z 625.741,A -85,B 0,C 180,E1 -30261.698,E2 -30261.698} C_VEL
LIN {X 0,Y 48.311,Z 627.469,A -85,B 0,C 180,E1 -30269.215,E2 -30269.215} C_VEL
LIN {X 0,Y 37.535,Z 627.694,A -85,B 0,C 180,E1 -30281.505,E2 -30281.505} C_VEL
LIN {X 0,Y 33.178,Z 627.205,A -85,B 0,C 180,E1 -30290.549,E2 -30290.549} C_VEL
LIN {X 0,Y 27.687,Z 625.06,A -85,B 0,C 180,E1 -30315.3,E2 -30315.3} C_VEL
LIN {X 0,Y 27.07,Z 623.39,A -85,B 0,C 180,E1 -30330.004,E2 -30330.004} C_VEL
LIN {X 0,Y 28.401,Z 619.965,A -85,B 0,C 180,E1 -30351.792,E2 -30351.792} C_VEL
LIN {X 0,Y 32.89,Z 615.428,A -85,B 0,C 180,E1 -30369.873,E2 -30369.873} C_VEL
LIN {X 0,Y 40.996,Z 608.519,A -85,B 0,C 180,E1 -30384.521,E2 -30384.521} C_VEL
LIN {X 0,Y 49.321,Z 600.996,A -85,B 0,C 180,E1 -30392.95,E2 -30392.95} C_VEL
LIN {X 0,Y 56.34,Z 593.715,A -85,B 0,C 180,E1 -30398.023,E2 -30398.023} C_VEL
LIN {X 0,Y 64.63,Z 583.926,A -85,B 0,C 180,E1 -30402.082,E2 -30402.082} C_VEL
LIN {X 0,Y 71.849,Z 573.439,A -85,B 0,C 180,E1 -30405.002,E2 -30405.002} C_VEL
LIN {X 0,Y 78.485,Z 561.861,A -85,B 0,C 180,E1 -30406.859,E2 -30406.859} C_VEL
LIN {X 0,Y 83.881,Z 549.59,A -85,B 0,C 180,E1 -30408.307,E2 -30408.307} C_VEL
LIN {X 0,Y 88.154,Z 536.305,A -85,B 0,C 180,E1 -30409.331,E2 -30409.331} C_VEL
